ORGANIZATION_BLOCK "SYS_OBNL_FLT"	// OB 85
TITLE = "Organization Block (OB) Not Loaded Fault"
//COPYRIGHT:    (C) 2000 BY  BUHLER LTD.
//                           CH-9240 UZWIL  SWITZERLAND
//
//PRODUCT:      PROJECT    
//
//TITLE:        Priority Class Error Organization Block (OB85)
//             
//
//--------------------------------------------------------------------------------
//
//IDENT:        AUTOR:              DEPT:                            DATE:
//STD_OB85.2.1  A.Egli              CT3                              23-Nov-2004
//              Only no stop when I/O access error updating the process image
//STD_OB85.2.0  A.Egli              CT3                              12-Jul-2004
//              LOG Message
//STD_OB85.1.0  A.Egli              CT3                              05-Nov-2002
//              1st Release
//
//--------------------------------------------------------------------------------
//
//PURPOSE:      
//
//RESTRICTIONS:
//
//--------------------------------------------------------------------------------
//
AUTHOR : EA
FAMILY : ASW
NAME : OBNLFLT
VERSION : 2.1
VAR_TEMP
  OB85_EV_CLASS : BYTE ;	//16#35 Event class 3
  OB85_FLT_ID : BYTE ;	//16#XX, Fault identification code
  OB85_PRIORITY : BYTE ;	//26 (Priority of 1 is lowest)
  OB85_OB_NUMBR : BYTE ;	//85 (Organization block 85, OB85)
  OB85_RESERVED_1 : BYTE ;	//Reserved for system
  OB85_RESERVED_2 : BYTE ;	//Reserved for system
  OB85_RESERVED_3 : INT ;	//Reserved for system
  OB85_ERR_EV_NUM : BYTE ;	//Number of event causing error
  OB85_ERR_EV_CLASS : BYTE ;	//Class of event causing error
  OB85_OB_PRIOR : BYTE ;	//Priority of OB causing error
  OB85_OB_NUM : BYTE ;	//Number of OB causing error
  OB85_DATE_TIME : DATE_AND_TIME ;	//Date and time OB85 started
  tmpHeader : WORD ;
  tmpObjNo : WORD ;	//OB-Nummer [80..121]
  EVClass_FLTID : WORD ;	//EV_Class / FLT_ID
  tmpPara3 : WORD ;
  tmpPara4 : WORD ;
  tmpPara5 : WORD ;
  tmpPara6 : WORD ;	//---
  tmpPara7 : WORD ;	//---
  tmpPara8 : WORD ;	//---
  tmpDate : WORD ;
  tmpYearMonth : WORD ;
  tmpDayHour : WORD ;
  tmpMinSec : WORD ;
  tmp_Z23 : DWORD ;
  tmpNoStop : BOOL ;
END_VAR
BEGIN
NETWORK
TITLE =
NETWORK
TITLE = Log Message: Header
//Header
      A(;
      L     #OB85_EV_CLASS;
      L     B#16#34;	// going
      ==I;
      );
      JCN   komm;
      L     3;
      JU    tran;
komm: L     1;	// coming
tran: SLW   5;
      +     11;	// NEW MessageFormatNo
      T     #tmpHeader;
NETWORK
TITLE = Log Message: Para1 = Object Number
//--System Message---
      L     85;
      T     #tmpObjNo;
NETWORK
TITLE = Log Message: Para2 to 11
////
//Para2: EV_Class / FLT_ID
      L     #OB85_FLT_ID;
      L     W#16#FF;	// Only Low Byte
      AW;
      L     #OB85_EV_CLASS;
      SLD   8;
      OW;
      T     #EVClass_FLTID;
//Para3: Depending on fault identification code
      L     #OB85_OB_NUMBR;
      T     #tmpPara3;
//Para4: DKZ23
      L     #OB85_RESERVED_1;
      T     #tmpPara4;
//Para5: Z1
      L     #OB85_RESERVED_3;
      T     #tmpPara5;
//Para6: Z23 HW
      LAR1  P##OB85_ERR_EV_NUM;
      L     LW [AR1,P#0.0];
      T     #tmpPara6;
//Para7: Z23 LW
      L     LW [AR1,P#2.0];
      T     #tmpPara7;
//Para9 to 11: Date/Time
      LAR1  P##OB85_DATE_TIME;
      L     LB [AR1,P#0.0];
      BTI;
      SLD   8;
      L     LB [AR1,P#1.0];
      BTI;
      OW;
      T     #tmpYearMonth;
      L     LB [AR1,P#2.0];
      BTI;
      SLD   8;
      L     LB [AR1,P#3.0];
      BTI;
      OW;
      T     #tmpDayHour;
      L     LB [AR1,P#4.0];
      BTI;
      SLD   8;
      L     LB [AR1,P#5.0];
      BTI;
      OW;
      T     #tmpMinSec;
NETWORK
TITLE = Faults without STOP
// // alle auskommentierten Einträge führen in STOP
//
//B1,B2,B3,B4: I/O access error when updating the process image
      A(;
      L     B#16#F0;
      L     #OB85_FLT_ID;
      AW;
      L     B#16#B0;
      ==I;
      );
      =     #tmpNoStop;
NETWORK
TITLE = Log Message: Entry
//Entre Log Message
      AN    #tmpNoStop;
      S     "SYS_LOG_Queue".CmdAddFastMsg;
      CALL  "SYS_LOG_EntryQueue" (
           DBNumber                 := 5,
           Header                   := #tmpHeader,
           Para1                    := #tmpObjNo,
           Para2                    := #EVClass_FLTID,
           Para3                    := #tmpPara3,
           Para4                    := #tmpPara4,
           Para5                    := #tmpPara5,
           Para6                    := #tmpPara6,
           Para7                    := #tmpPara7,
           Para8                    := W#16#0,
           Para9                    := #tmpYearMonth,
           Para10                   := #tmpDayHour,
           Para11                   := #tmpMinSec);	//Header / Para1: ObjectNo / Para2: Class / FLTID / Para3: OB Number / Para4: DKZ23 / Para5: Z1 / Para6: Z23 HW / Para7: Z23 LW / Para8:  / Para9:  Year / Month / Para10: Day  / Hour / Para11: Min  / Sec 
NETWORK
TITLE = Stop PLC
      A     #tmpNoStop;
      BEC;
//**********************
// Bring CPU to Stop
      CALL  "SIEMENS_STP";
//**********************
NETWORK
TITLE = End of block
      BE;
END_ORGANIZATION_BLOCK

ORGANIZATION_BLOCK "SYS_RACK_FLT"	// OB 86
TITLE = "Loss Of Rack Fault"
//COPYRIGHT:    (C) 2000 BY  BUHLER AG
//                           CH-9240 UZWIL  SWITZERLAND
//
//PRODUCT:      PROJECT
//
//TITLE:        Loss of rack fault
//               Extended rack faults
//               DP-Master or slave faults
//              Erweiterungsgerätanschaltungsfehler
//               Erweiterungsgerätefehler
//               Profibus-DB Master- und Slavefehler
//
//--------------------------------------------------------------------------------
//IDENT:        AUTHOR:             DEPT:                             DATE:
//
//Pxx_OB086.2.0 A.Egli              CT3                               12-Jul-2004
//              Log message added
//Pxx_OB086.1.0 Ph. Engler          MU664                             16-Jan-2002
//              1st Release
//
//--------------------------------------------------------------------------------
//
//PURPOSE:      
//
//RESTRICTIONS: 
//
//--------------------------------------------------------------------------------
//
AUTHOR : EA
FAMILY : ASW
NAME : RACKFLT
VERSION : 2.0
VAR_TEMP
  OB86_EV_CLASS : BYTE ;	//16#38/39 Event class 3
  OB86_FLT_ID : BYTE ;	//16#C1/C4/C5, Fault identification code
  OB86_PRIORITY : BYTE ;	//26/28 (Priority of 1 is lowest)
  OB86_OB_NUMBR : BYTE ;	//86 (Organization block 86, OB86)
  OB86_RESERVED_1 : BYTE ;	//Reserved for system
  OB86_RESERVED_2 : BYTE ;	//Reserved for system
  OB86_MDL_ADDR : WORD ;	//Depending on fault identification code
  OB86_RACKS_FLTD : ARRAY  [0 .. 31 ] OF BOOL ;	//Racks in fault
  OB86_DATE_TIME : DATE_AND_TIME ;	//Date and time OB86 started
  tmpHeader : WORD ;
  tmpObjNo : WORD ;	//OB-Nummer [80..121]
  EVClass_FLTID : WORD ;	//EV_Class / FLT_ID
  tmpPara3 : WORD ;	//
  tmpPara4 : WORD ;	//
  tmpPara5 : WORD ;	//
  tmpPara6 : WORD ;	//
  tmpPara7 : WORD ;	//
  tmpDate : WORD ;
  tmpYearMonth : WORD ;
  tmpDayHour : WORD ;
  tmpMinSec : WORD ;
  tmp_Z23 : DWORD ;
  tmpSlave : INT ;
  tmpMaster : INT ;
  tmpNoStop : BOOL ;
END_VAR
BEGIN
NETWORK
TITLE = Detailed Diagnosis in OB86 (interrupt)
      CALL  "SYS_DPDiagMain";
NETWORK
TITLE = Log Message: Header
//Header
      A(;
      L     #OB86_EV_CLASS;
      L     B#16#38;	// going
      ==I;
      );
      JCN   komm;
      L     3;
      JU    tran;
komm: L     1;	// coming
tran: SLW   5;
      +     11;	// NEW MessageFormatNo
      T     #tmpHeader;
NETWORK
TITLE = Log Message: Para1 = Object Number
//Para1: Object Number
      LAR1  P##OB86_RACKS_FLTD;
      L     LD [AR1,P#0.0];
      T     #tmp_Z23;
      L     #tmp_Z23;
      SRD   8;
      L     DW#16#FF;
      AW;
      L     1000;
      *I;
      T     #tmpMaster;
      L     #tmp_Z23;
      L     DW#16#FF;
      AW;
      T     #tmpSlave;
//--DP Rack -----
      L     #OB86_FLT_ID;
      L     B#16#C1;
      ==I;
      JC    OJRA;
      L     #OB86_FLT_ID;
      L     B#16#C2;
      ==I;
      JC    OJRA;
      L     #OB86_FLT_ID;
      L     B#16#C6;
      ==I;
      JC    OJRA;
      JU    OJC3;
OJRA: LAR1  P##OB86_RACKS_FLTD;
//    Check Bit 1..21 of OB86_Racks_FLTD
      L     10001;
      T     #tmpObjNo;
OJR2: A     L [AR1,P#0.1];
      JC    OJJO;
      +AR1  P#0.1;
      L     121;
      L     #tmpObjNo;
      <=I;
      JC    OJR2;
      JU    OJSM;	//-->Illegal RackNr-->  Print as System message
//--DP Master -----
OJC3: L     #OB86_FLT_ID;
      L     B#16#C3;
      ==I;
      JC    OJMA;
      JU    OJC4;
OJMA: L     #tmpMaster;
      T     #tmpObjNo;
      JU    OJJO;
//---DP Station----
OJC4: L     #OB86_FLT_ID;
      L     B#16#C4;
      ==I;
      JC    OJSL;
      L     #OB86_FLT_ID;
      L     B#16#C5;
      ==I;
      JC    OJSL;
      L     #OB86_FLT_ID;
      L     B#16#C7;
      ==I;
      JC    OJSL;
      L     #OB86_FLT_ID;
      L     B#16#C8;
      ==I;
      JC    OJSL;
      JU    OJSM;
OJSL: L     #tmpMaster;
      L     #tmpSlave;
      +I;
      T     #tmpObjNo;
      JU    OJJO;
//--System Message---
OJSM: L     86;
      T     #tmpObjNo;
OJJO: NOP   0;
NETWORK
TITLE = Log Message: Para2 to 11
////
//Para2: EV_Class / FLT_ID
      L     #OB86_FLT_ID;
      L     W#16#FF;	// Only Low Byte
      AW;
      L     #OB86_EV_CLASS;
      SLD   8;
      OW;
      T     #EVClass_FLTID;
//Para3: Depending on fault identification code
      L     #OB86_OB_NUMBR;
      T     #tmpPara3;
//Para4:not used
      L     0;
      T     #tmpPara4;
//Para5: MDL_ADDR
      L     #OB86_MDL_ADDR;
      T     #tmpPara5;
//Para6: Z23 HW
      LAR1  P##OB86_RACKS_FLTD;
      L     LW [AR1,P#0.0];
      T     #tmpPara6;
//Para7: Z23 LW
      L     LW [AR1,P#2.0];
      T     #tmpPara7;
//Para9 to 11: Date/Time
      LAR1  P##OB86_DATE_TIME;
      L     LB [AR1,P#0.0];
      BTI;
      SLD   8;
      L     LB [AR1,P#1.0];
      BTI;
      OW;
      T     #tmpYearMonth;
      L     LB [AR1,P#2.0];
      BTI;
      SLD   8;
      L     LB [AR1,P#3.0];
      BTI;
      OW;
      T     #tmpDayHour;
      L     LB [AR1,P#4.0];
      BTI;
      SLD   8;
      L     LB [AR1,P#5.0];
      BTI;
      OW;
      T     #tmpMinSec;
NETWORK
TITLE = Faults without STOP
// // alle auskommentierten Einträge führen in STOP
//
// C1 Expansion rack failure
      O(;
      L     #OB86_FLT_ID;
      L     B#16#C1;	// 
      ==I;
      );
// C2 Expansion rack operational again
      O(;
      L     #OB86_FLT_ID;
      L     B#16#C2;	// 
      ==I;
      );
// C3 Failure of  DP master
      O(;
      L     #OB86_FLT_ID;
      L     B#16#C3;	// 
      ==I;
      );
// C4 Failure of DP Slave
      O(;
      L     #OB86_FLT_ID;
      L     B#16#C4;	// 
      ==I;
      );
// C5 Fault in a DP Slave
      O(;
      L     #OB86_FLT_ID;
      L     B#16#C5;	// 
      ==I;
      );
// C6 Expansion rack with error in module parameter
      O(;
      L     #OB86_FLT_ID;
      L     B#16#C6;	// 
      ==I;
      );
// C7 Return DP Slave with error in modul parameter
      O(;
      L     #OB86_FLT_ID;
      L     B#16#C7;	// 
      ==I;
      );
// C8 DP Slave configuartion <> actual configuration
      O(;
      L     #OB86_FLT_ID;
      L     B#16#C8;	// 
      ==I;
      );
      =     #tmpNoStop;
NETWORK
TITLE = Log Message: Entry
//Entre Log Message
      AN    #tmpNoStop;
      S     "SYS_LOG_Queue".CmdAddFastMsg;
      CALL  "SYS_LOG_EntryQueue" (
           DBNumber                 := 5,
           Header                   := #tmpHeader,
           Para1                    := #tmpObjNo,
           Para2                    := #EVClass_FLTID,
           Para3                    := #tmpPara3,
           Para4                    := W#16#0,
           Para5                    := #tmpPara5,
           Para6                    := #tmpPara6,
           Para7                    := #tmpPara7,
           Para8                    := W#16#0,
           Para9                    := #tmpYearMonth,
           Para10                   := #tmpDayHour,
           Para11                   := #tmpMinSec);	//Header / Para1: ObjectNo / Para2: Class / FLTID / Para3: OB Number / Para4: / Para5: MDL_ADDR / Para6: Z23 HW / Para7: Z23 HW / Para8:  / Para9:  Year / Month / Para10: Day  / Hour / Para11: Min  / Sec 
NETWORK
TITLE = Stop PLC
      A     #tmpNoStop;
      BEC;
//**********************
// Bring CPU to Stop
      CALL  "SIEMENS_STP";
//**********************
NETWORK
TITLE = End of block
      BE;
END_ORGANIZATION_BLOCK

ORGANIZATION_BLOCK "PLC_StUpNewstart"	// OB 100
TITLE = Startup program on newstart
//COPYRIGHT:    (C) 2000 BY  BUHLER AG
//                           CH-9240 UZWIL  SWITZERLAND
//
//PRODUCT:      PROJECT
//
//TITLE:        Startup program on newstart
//              
//              Anlaufprogramm bei Neustart
//
//
//--------------------------------------------------------------------------------
//
//IDENT:        AUTHOR:             DEPT:                             DATE:
//
//Pxx_OB102.2.0 A.Egli              CT3                               15-Jul-2004
//              Log Message
//Pxx_OB100.1.0 Ph. Engler          MU664                             05-Jan-2000
//              1st Release
//
//--------------------------------------------------------------------------------
//
//PURPOSE:      
//
//RESTRICTIONS: 
//
//--------------------------------------------------------------------------------
//
AUTHOR : PE
FAMILY : ASW
NAME : StUpNew
VERSION : 2.0
VAR_TEMP
  OB100_EV_CLASS : BYTE ;	//16#13, Event class 1, Entering event state, Event logged in diagnostic buffer
  OB100_STRTUP : BYTE ;	//16#81/82/83/84 Method of startup
  OB100_PRIORITY : BYTE ;	//27 (Priority of 1 is lowest)
  OB100_OB_NUMBR : BYTE ;	//100 (Organization block 100, OB100)
  OB100_RESERVED_1 : BYTE ;	//Reserved for system
  OB100_RESERVED_2 : BYTE ;	//Reserved for system
  OB100_STOP : WORD ;	//Event that caused CPU to stop (16#4xxx)
  OB100_STRT_INFO : DWORD ;	//Information on how system started
  OB100_DATE_TIME : DATE_AND_TIME ;	//Date and time OB100 started
  tmpHeader : WORD ;
  tmpObjNo : WORD ;	//OB-Nummer [80..121]
  EVClass_FLTID : WORD ;	//EV_Class / FLT_ID
  tmpPara3 : WORD ;	//
  tmpDate : WORD ;
  tmpYearMonth : WORD ;
  tmpDayHour : WORD ;
  tmpMinSec : WORD ;
END_VAR
BEGIN
NETWORK
TITLE = Create startup signals
      L     #OB100_STRTUP;
      L     B#16#81;
      ==I;
      S     "PLC_SystemDB".Startup.CmdNewstartMan;
      L     #OB100_STRTUP;
      L     B#16#82;
      ==I;
      S     "PLC_SystemDB".Startup.CmdNewstartAuto;
NETWORK
TITLE = Startup counters
      AN    "PLC_SystemDB".Startup.CmdNewstartMan;
      JC    n2n1;
      L     "PLC_SystemDB".StartupCounter.NewstartMan;
      +     1;
      T     "PLC_SystemDB".StartupCounter.NewstartMan;
      JU    n2e;
n2n1: AN    "PLC_SystemDB".Startup.CmdNewstartAuto;
      JC    n2e;
      L     "PLC_SystemDB".StartupCounter.NewstartAuto;
      +     1;
      T     "PLC_SystemDB".StartupCounter.NewstartAuto;
n2e:  NOP   0;
NETWORK
TITLE = General plc startup functions
      CALL  "SYS_GeneralPLCStartup";
NETWORK
TITLE = Special plant startup functions
NETWORK
TITLE = Reset startup flags
      SET;
      R     "PLC_SystemDB".Startup.CmdNewstartMan;
      R     "PLC_SystemDB".Startup.CmdNewstartAuto;
NETWORK
TITLE = Log Message: Header
//Header
      L     3;	// Operator
      SLW   5;
      +     11;	// NEW MessageFormatNo
      T     #tmpHeader;
NETWORK
TITLE = Log Message: Para1 = Object Number
//Para1: Object Number
//--System Message---
      L     #OB100_OB_NUMBR;
      T     #tmpObjNo;
NETWORK
TITLE = Log Message: Para2 to 11
////
//Para2: EV_Class / FLT_ID
      L     #OB100_STRTUP;
      L     W#16#FF;	// Only Low Byte
      AW;
      L     #OB100_EV_CLASS;
      SLD   8;
      OW;
      T     #EVClass_FLTID;
//Para3: Depending on fault identification code
      L     #OB100_OB_NUMBR;
      T     #tmpPara3;
//Para9 to 11: Date/Time
      LAR1  P##OB100_DATE_TIME;
      L     LB [AR1,P#0.0];
      BTI;
      SLD   8;
      L     LB [AR1,P#1.0];
      BTI;
      OW;
      T     #tmpYearMonth;
      L     LB [AR1,P#2.0];
      BTI;
      SLD   8;
      L     LB [AR1,P#3.0];
      BTI;
      OW;
      T     #tmpDayHour;
      L     LB [AR1,P#4.0];
      BTI;
      SLD   8;
      L     LB [AR1,P#5.0];
      BTI;
      OW;
      T     #tmpMinSec;
NETWORK
TITLE = Log Message: Entry
//Entre Log Message
      CALL  "SYS_LOG_EntryQueue" (
           DBNumber                 := 5,
           Header                   := #tmpHeader,
           Para1                    := #tmpObjNo,
           Para2                    := #EVClass_FLTID,
           Para3                    := #tmpPara3,
           Para4                    := W#16#0,
           Para5                    := W#16#0,
           Para6                    := W#16#0,
           Para7                    := W#16#0,
           Para8                    := W#16#0,
           Para9                    := #tmpYearMonth,
           Para10                   := #tmpDayHour,
           Para11                   := #tmpMinSec);	//Header / Para1: ObjectNo / Para2: Class / STRTUP / Para3: OB Number / Para4: / Para5:  / Para6:  / Para7: / Para8:  / Para9:  Year / Month / Para10: Day  / Hour / Para11: Min  / Sec 
NETWORK
TITLE = End of block
      BE;
END_ORGANIZATION_BLOCK

ORGANIZATION_BLOCK "PLC_StUpRestart"	// OB 101
TITLE = Startup program on restart
//COPYRIGHT:    (C) 2000 BY  BUHLER AG
//                           CH-9240 UZWIL  SWITZERLAND
//
//PRODUCT:      PROJECT
//
//TITLE:        Startup program on restart
//                 After voltage returned
//              Anlaufprogramm  bei Wiederanlauf
//                 Nach Spannungswiederkehr
//
//--------------------------------------------------------------------------------
//
//IDENT:        AUTHOR:             DEPT:                             DATE:
//
//Pxx_OB101.3.0 A.Egli              CT3                               15-Jul-2004
//              The following lines are moved to OB1
//                R     "PLC_SystemDB".Startup.CmdRestartMan
//                R     "PLC_SystemDB".Startup.CmdRestartAuto
//Pxx_OB101.2.0 A.Egli              CT3                               15-Jul-2004
//              Log Message
//Pxx_OB101.1.0 Ph. Engler          MU664                             05-Jan-2000
//              1st Release
//
//--------------------------------------------------------------------------------
//
//PURPOSE:      
//
//RESTRICTIONS: 
//
//--------------------------------------------------------------------------------
//
AUTHOR : PE
FAMILY : ASW
NAME : StUpRest
VERSION : 3.0
VAR_TEMP
  OB101_EV_CLASS : BYTE ;	//16#13, Event class 1, Entering event state, Event logged in diagnostic buffer
  OB101_STRTUP : BYTE ;	//16#81/82/83/84 Method of startup
  OB101_PRIORITY : BYTE ;	//27 (Priority of 1 is lowest)
  OB101_OB_NUMBR : BYTE ;	//101 (Organization block 101, OB101)
  OB101_RESERVED_1 : BYTE ;	//Reserved for system
  OB101_RESERVED_2 : BYTE ;	//Reserved for system
  OB101_STOP : WORD ;	//Event that caused CPU to stop (16#4xxx)
  OB101_STRT_INFO : DWORD ;	//Information on how system started
  OB101_DATE_TIME : DATE_AND_TIME ;	//Date and time OB101 started
  tmpHeader : WORD ;
  tmpObjNo : WORD ;	//OB-Nummer [80..121]
  EVClass_FLTID : WORD ;	//EV_Class / FLT_ID
  tmpPara3 : WORD ;	//
  tmpDate : WORD ;
  tmpYearMonth : WORD ;
  tmpDayHour : WORD ;
  tmpMinSec : WORD ;
END_VAR
BEGIN
NETWORK
TITLE = Create startup flags
      L     #OB101_STRTUP;
      L     B#16#83;
      ==I;
      S     "PLC_SystemDB".Startup.CmdRestartMan;
      L     #OB101_STRTUP;
      L     B#16#84;
      ==I;
      S     "PLC_SystemDB".Startup.CmdRestartAuto;
NETWORK
TITLE = Startup counters
      AN    "PLC_SystemDB".Startup.CmdRestartMan;
      JC    n2n1;
      L     "PLC_SystemDB".StartupCounter.RestartMan;
      +     1;
      T     "PLC_SystemDB".StartupCounter.RestartMan;
      JU    n2e;
n2n1: AN    "PLC_SystemDB".Startup.CmdRestartAuto;
      JC    n2e;
      L     "PLC_SystemDB".StartupCounter.RestartAuto;
      +     1;
      T     "PLC_SystemDB".StartupCounter.RestartAuto;
n2e:  NOP   0;
NETWORK
TITLE = General plc startup functions
      CALL  "SYS_GeneralPLCStartup";
NETWORK
TITLE = Special plant startup functions
NETWORK
TITLE = Reset startup flags
//[3.0]      SET   
//[3.0]      R     "PLC_SystemDB".Startup.CmdRestartMan
//[3.0]      R     "PLC_SystemDB".Startup.CmdRestartAuto
NETWORK
TITLE = Log Message: Header
//Header
      L     3;	// Operator
      SLW   5;
      +     11;	// NEW MessageFormatNo
      T     #tmpHeader;
NETWORK
TITLE = Log Message: Para1 = Object Number
//Para1: Object Number
//--System Message---
      L     #OB101_OB_NUMBR;
      T     #tmpObjNo;
NETWORK
TITLE = Log Message: Para2 to 11
////
//Para2: EV_Class / FLT_ID
      L     #OB101_STRTUP;
      L     W#16#FF;	// Only Low Byte
      AW;
      L     #OB101_EV_CLASS;
      SLD   8;
      OW;
      T     #EVClass_FLTID;
//Para3: Depending on fault identification code
      L     #OB101_OB_NUMBR;
      T     #tmpPara3;
//Para9 to 11: Date/Time
      LAR1  P##OB101_DATE_TIME;
      L     LB [AR1,P#0.0];
      BTI;
      SLD   8;
      L     LB [AR1,P#1.0];
      BTI;
      OW;
      T     #tmpYearMonth;
      L     LB [AR1,P#2.0];
      BTI;
      SLD   8;
      L     LB [AR1,P#3.0];
      BTI;
      OW;
      T     #tmpDayHour;
      L     LB [AR1,P#4.0];
      BTI;
      SLD   8;
      L     LB [AR1,P#5.0];
      BTI;
      OW;
      T     #tmpMinSec;
NETWORK
TITLE = Log Message: Entry
//Entre Log Message
      CALL  "SYS_LOG_EntryQueue" (
           DBNumber                 := 5,
           Header                   := #tmpHeader,
           Para1                    := #tmpObjNo,
           Para2                    := #EVClass_FLTID,
           Para3                    := #tmpPara3,
           Para4                    := W#16#0,
           Para5                    := W#16#0,
           Para6                    := W#16#0,
           Para7                    := W#16#0,
           Para8                    := W#16#0,
           Para9                    := #tmpYearMonth,
           Para10                   := #tmpDayHour,
           Para11                   := #tmpMinSec);	//Header / Para1: ObjectNo / Para2: Class / STRTUP / Para3: OB Number / Para4: / Para5:  / Para6:  / Para7: / Para8:  / Para9:  Year / Month / Para10: Day  / Hour / Para11: Min  / Sec 
NETWORK
TITLE = End of block
      BE;
END_ORGANIZATION_BLOCK

ORGANIZATION_BLOCK "PLC_StUpColdstart"	// OB 102
TITLE = Startup program on coldstart
//COPYRIGHT:    (C) 2000 BY  BUHLER AG
//                           CH-9240 UZWIL  SWITZERLAND
//
//PRODUCT:      PROJECT
//
//TITLE:        Startup program on coldstart
//              
//              Anlaufprogramm bei Kaltstart
//
//
//--------------------------------------------------------------------------------
//
//IDENT:        AUTHOR:             DEPT:                             DATE:
//
//Pxx_OB102.2.0 A.Egli              CT3                               15-Jul-2004
//              Log Message
//Pxx_OB102.1.0 Ph. Engler          MU664                             17-Dez-2000
//              1st Release
//
//--------------------------------------------------------------------------------
//
//PURPOSE:      
//
//RESTRICTIONS: 
//
//--------------------------------------------------------------------------------
//
AUTHOR : PE
FAMILY : ASW
NAME : StUpCold
VERSION : 2.0
VAR_TEMP
  OB102_EV_CLASS : BYTE ;	//16#13, Event class 1, Entering event state, Event logged in diagnostic buffer
  OB102_STRTUP : BYTE ;	//16#85...8B Method of startup
  OB102_PRIORITY : BYTE ;	//27 (Priority of 1 is lowest)
  OB102_OB_NUMBR : BYTE ;	//102 (Organization block 102, OB102)
  OB102_RESERVED_1 : BYTE ;	//Reserved for system
  OB102_RESERVED_2 : BYTE ;	//Reserved for system
  OB102_STOP : WORD ;	//Event that caused CPU to stop (16#4xxx)
  OB102_STRT_INFO : DWORD ;	//Information on how system started
  OB102_DATE_TIME : DATE_AND_TIME ;	//Date and time OB102 started
  tmpHeader : WORD ;
  tmpObjNo : WORD ;	//OB-Nummer [80..121]
  EVClass_FLTID : WORD ;	//EV_Class / FLT_ID
  tmpPara3 : WORD ;	//
  tmpDate : WORD ;
  tmpYearMonth : WORD ;
  tmpDayHour : WORD ;
  tmpMinSec : WORD ;
END_VAR
BEGIN
NETWORK
TITLE = Create startup signals
      L     #OB102_STRTUP;
      L     B#16#85;
      ==I;
      S     "PLC_SystemDB".Startup.CmdColdstartMan;
// 
      L     #OB102_STRTUP;
      L     B#16#86;
      ==I;
      S     "PLC_SystemDB".Startup.CmdColdstartAuto;
NETWORK
TITLE = Startup counters
      AN    "PLC_SystemDB".Startup.CmdColdstartMan;
      JC    n2n1;
      L     "PLC_SystemDB".StartupCounter.ColdstartMan;
      +     1;
      T     "PLC_SystemDB".StartupCounter.ColdstartMan;
      JU    n2e;
n2n1: AN    "PLC_SystemDB".Startup.CmdColdstartAuto;
      JC    n2e;
      L     "PLC_SystemDB".StartupCounter.ColdstartAuto;
      +     1;
      T     "PLC_SystemDB".StartupCounter.ColdstartAuto;
n2e:  NOP   0;
NETWORK
TITLE = General plc startup functions
      CALL  "SYS_GeneralPLCStartup";
NETWORK
TITLE = Special plant startup functions
NETWORK
TITLE = Reset startup flags
      SET;
      R     "PLC_SystemDB".Startup.CmdColdstartMan;
      R     "PLC_SystemDB".Startup.CmdColdstartAuto;
NETWORK
TITLE = Log Message: Header
//Header
      L     3;	// Operator
      SLW   5;
      +     11;	// NEW MessageFormatNo
      T     #tmpHeader;
NETWORK
TITLE = Log Message: Para1 = Object Number
//Para1: Object Number
//--System Message---
      L     #OB102_OB_NUMBR;
      T     #tmpObjNo;
NETWORK
TITLE = Log Message: Para2 to 11
////
//Para2: EV_Class / FLT_ID
      L     #OB102_STRTUP;
      L     W#16#FF;	// Only Low Byte
      AW;
      L     #OB102_EV_CLASS;
      SLD   8;
      OW;
      T     #EVClass_FLTID;
//Para3: Depending on fault identification code
      L     #OB102_OB_NUMBR;
      T     #tmpPara3;
//Para9 to 11: Date/Time
      LAR1  P##OB102_DATE_TIME;
      L     LB [AR1,P#0.0];
      BTI;
      SLD   8;
      L     LB [AR1,P#1.0];
      BTI;
      OW;
      T     #tmpYearMonth;
      L     LB [AR1,P#2.0];
      BTI;
      SLD   8;
      L     LB [AR1,P#3.0];
      BTI;
      OW;
      T     #tmpDayHour;
      L     LB [AR1,P#4.0];
      BTI;
      SLD   8;
      L     LB [AR1,P#5.0];
      BTI;
      OW;
      T     #tmpMinSec;
NETWORK
TITLE = Log Message: Entry
//Entre Log Message
      CALL  "SYS_LOG_EntryQueue" (
           DBNumber                 := 5,
           Header                   := #tmpHeader,
           Para1                    := #tmpObjNo,
           Para2                    := #EVClass_FLTID,
           Para3                    := #tmpPara3,
           Para4                    := W#16#0,
           Para5                    := W#16#0,
           Para6                    := W#16#0,
           Para7                    := W#16#0,
           Para8                    := W#16#0,
           Para9                    := #tmpYearMonth,
           Para10                   := #tmpDayHour,
           Para11                   := #tmpMinSec);	//Header / Para1: ObjectNo / Para2: Class / STRTUP / Para3: OB Number / Para4: / Para5:  / Para6:  / Para7: / Para8:  / Para9:  Year / Month / Para10: Day  / Hour / Para11: Min  / Sec 
NETWORK
TITLE = End of block
      BE;
END_ORGANIZATION_BLOCK

ORGANIZATION_BLOCK "SYS_PROG_ERR"	// OB 121
//COPYRIGHT:    (C) 2000 BY  BUHLER AG
//                           CH-9240 UZWIL  SWITZERLAND
//
//PRODUCT:      PROJECT
//
//TITLE:        OB121 
//              
//
//--------------------------------------------------------------------------------
//IDENT:        AUTHOR:             DEPT:                             DATE:
//
//OB121.2.0     A.Egli              CT3                               13-Jul-2004
//              1st Release
//OB121.1A      TIK                 MU664                             13-Apr-99
//              1st Release
//OB121.1B      Tho                 FU53                              16-Dez-99
//              FU-Version erstellt 
//
//--------------------------------------------------------------------------------
//
//PURPOSE:      
//
//RESTRICTIONS: 
//
//--------------------------------------------------------------------------------
//
AUTHOR : EA
FAMILY : ASW
NAME : PROG_ERR
VERSION : 2.0
VAR_TEMP
  OB121_EV_CLASS : BYTE ;	//16#25, Event class 2, Entering event state, Internal fault event
  OB121_SW_FLT : BYTE ;	//16#XX Software programming fault
  OB121_PRIORITY : BYTE ;	//X = Priority of OB where fault occured (Priority of 1 is lowest)
  OB121_OB_NUMBR : BYTE ;	//121 (Organization block 121, OB121)
  OB121_BLK_TYPE : BYTE ;	//16#88/8A/8B/8C/8E Type of block fault occured in
  OB121_RESERVED_1 : BYTE ;	//Reserved for system
  OB121_FLT_REG : WORD ;	//16#XX Specific register that caused fault
  OB121_BLK_NUM : WORD ;	//Number of block that programming fault occured in
  OB121_PRG_ADDR : WORD ;	//Address in block where programming fault occured
  OB121_DATE_TIME : DATE_AND_TIME ;	//Date and time OB121 started
  tmpHeader : WORD ;
  tmpObjNo : WORD ;	//OB-Nummer [80..121]
  EVClass_FLTID : WORD ;	//EV_Class / FLT_ID
  tmpPara3 : WORD ;	//Reserved 1 for system
  tmpPara4 : WORD ;	//Input module (01010100), Output module (01010101)
  tmpPara5 : WORD ;	//Base address of module with point fault
  tmpPara6 : WORD ;	//Module type with point fault
  tmpPara7 : WORD ;	//Module type with point fault
  tmpYearMonth : WORD ;
  tmpDayHour : WORD ;
  tmpMinSec : WORD ;
  tmpNoStop : BOOL ;
END_VAR
BEGIN
NETWORK
TITLE =
NETWORK
TITLE = Log Message: Header
      A(;
      L     #OB121_EV_CLASS;
      L     B#16#38;	// going
      ==I;
      );
      JCN   komm;
      L     3;
      JU    tran;
komm: L     1;	// coming
tran: SLW   5;
      +     11;	// NEW MessageFormatNo
      T     #tmpHeader;
NETWORK
TITLE = Log Message: Para1 = Object Number
//--System Message---
      L     121;
      T     #tmpObjNo;
NETWORK
TITLE = Log Message: Para2 to 11
////
//Para2: EV_Class / FLT_ID
      L     #OB121_SW_FLT;
      L     W#16#FF;	// Only Low Byte
      AW;
      L     #OB121_EV_CLASS;
      SLD   8;
      OW;
      T     #EVClass_FLTID;
//Para3: OB_NUMBR
      L     #OB121_OB_NUMBR;
      T     #tmpPara3;
//Para4: OB121_FLT_REG
      L     #OB121_FLT_REG;
      T     #tmpPara4;
//Para5: OB121_BLK_TYPE
      L     #OB121_BLK_TYPE;
      T     #tmpPara5;
//Para6: Number of block that programming fault occured in
      L     #OB121_BLK_NUM;
      T     #tmpPara6;
//Para7: Address in block where programming fault occured
      L     #OB121_PRG_ADDR;
      T     #tmpPara7;
//Para9 to 11: Date/Time
      LAR1  P##OB121_DATE_TIME;
      L     LB [AR1,P#0.0];
      BTI;
      SLD   8;
      L     LB [AR1,P#1.0];
      BTI;
      OW;
      T     #tmpYearMonth;
      L     LB [AR1,P#2.0];
      BTI;
      SLD   8;
      L     LB [AR1,P#3.0];
      BTI;
      OW;
      T     #tmpDayHour;
      L     LB [AR1,P#4.0];
      BTI;
      SLD   8;
      L     LB [AR1,P#5.0];
      BTI;
      OW;
      T     #tmpMinSec;
NETWORK
TITLE = Faults without STOP
//// alle auskommentierten Einträge führen in STOP 
//
      CLR;	//init.VKE  
// 21 BCD conversion error
      O(;
      L     #OB121_SW_FLT;
      L     B#16#21;	// 
      ==I;
      );
// 22 Area length error when reading
//      O(    
//      L     #OB121_SW_FLT
//      L     B#16#22                     // 
//      ==I   
//      )     
// 23 Range error when writing
//      O(    
//      L     #OB121_SW_FLT
//      L     B#16#23                     // 
//      ==I   
//      )     
// 24 Range access with pointer
//      O(    
//      L     #OB121_SW_FLT
//      L     B#16#24                     // 
//      ==I   
//      )     
// 25 Writing access with pointer
//      O(    
//      L     #OB121_SW_FLT
//      L     B#16#25                     // 
//      ==I   
//      )     
// 26 Error for timer number
//     O(    
//      L     #OB121_SW_FLT
//      L     B#16#26                     // 
//      ==I   
//      )     
// 27 Error for Counter
//      O(           
//      L     #OB121_SW_FLT
//      L     B#16#27                     // 
//      ==I   
//      )     
// 28  Reading access with pointer Bit<>0
//      O(    
//      L     #OB121_SW_FLT
//      L     B#16#28                     // 
//      ==I   
//      )     
// 29  Reading access with pointer Bit<>0
//      O(    
//      L     #OB121_SW_FLT
//      L     B#16#29                     // 
//      ==I   
//      )     
// 30 Write access GlobalDB
//      O(    
//      L     #OB121_SW_FLT
//      L     B#16#30                     // 
//      ==I   
//      )     
// 31 Write access InstanzDB
//      O(    
//      L     #OB121_SW_FLT
//      L     B#16#31                     // 
//     ==I   
//     )     
// 32 DB number GlobalDB
//      O(    
//      L     #OB121_SW_FLT
//      L     B#16#32                     // 
//      ==I   
//      )     
// 33 DB number InstanzDB
//      O(    
//      L     #OB121_SW_FLT
//      L     B#16#33                     // 
//      ==I   
//      )     
// 34 FC Number
//      O(    
//      L     #OB121_SW_FLT
//      L     B#16#34                     // 
//      ==I   
//      )     
// 35 FB Number
//      O(    
//      L     #OB121_SW_FLT
//      L     B#16#35                     // 
//      ==I   
//      )     
// 3A DB not loaded
//      O(    
//      L     #OB121_SW_FLT
//      L     B#16#3A                     // 
//      ==I   
//      )     
// 3C FC not loaded
//      O(    
//      L     #OB121_SW_FLT
//      L     B#16#3C                     // 
//      ==I   
//      )     
// 3D SFC not loaded
//      O(    
//      L     #OB121_SW_FLT
//      L     B#16#3D                     // 
//      ==I   
//      )     
// 3E FB not loaded
//      O(    
//      L     #OB121_SW_FLT
//      L     B#16#3E                     // 
//      ==I   
//      )     
// 3F SFB not loaded
//      O(    
//      L     #OB121_SW_FLT
//      L     B#16#3F                     // 
//      ==I   
//      )     
      =     #tmpNoStop;
NETWORK
TITLE = Log Message: Entry
//Log Meldung eintragen
      L     "SYS_LOG_Queue".VarNrOfMsgInQueue;
      L     0;
      <>I;
      A     #tmpNoStop;
      JC    LOJ0;
      AN    #tmpNoStop;
      S     "SYS_LOG_Queue".CmdAddFastMsg;
      CALL  "SYS_LOG_EntryQueue" (
           DBNumber                 := 5,
           Header                   := #tmpHeader,
           Para1                    := #tmpObjNo,
           Para2                    := #EVClass_FLTID,
           Para3                    := #tmpPara3,
           Para4                    := #tmpPara4,
           Para5                    := #tmpPara5,
           Para6                    := #tmpPara6,
           Para7                    := #tmpPara7,
           Para8                    := W#16#0,
           Para9                    := #tmpYearMonth,
           Para10                   := #tmpDayHour,
           Para11                   := #tmpMinSec);	//Header / Para1: ObjectNo / Para2: Class / FLTID / Para3: OB Number / Para4: FLT_REG / Para5: BLK_TYPE / Para6: BLK_NUM / Para7: PGR_ADDR / Para8:  / Para9:  Year / Month / Para10: Day  / Hour / Para11: Min  / Sec 
LOJ0: NOP   0;
NETWORK
TITLE = Stop PLC
      A     #tmpNoStop;
      BEC;
//**********************
// Bring CPU to Stop
      CALL  "SIEMENS_STP";
//**********************
NETWORK
TITLE = End of block
      BE;
END_ORGANIZATION_BLOCK

ORGANIZATION_BLOCK "SYS_MOD_ERR"	// OB 122
TITLE = "Module Access Error"
//COPYRIGHT:    (C) 2000 BY  BUHLER AG
//                           CH-9240 UZWIL  SWITZERLAND
//
//PRODUCT:      GEN_MU664
//
//TITLE:        Failure reading/wrinting to/from the peripherie
//
//              Peripheriezugriffsfehler
//              
//
//--------------------------------------------------------------------------------
//IDENT:        AUTHOR:             DEPT:                              DATE:
//
//GEN_OB122.2.0 Ph. Engler          MU664                              11-Feb-2003
//              Redesign GCS7 Release 2
//GEN_OB122.1.1 Ph. Engler          MU664                              22-Oct-2002
//              - MU test flag integrated
//GEN_OB122.1.0 A. Egli             CT3                                19-Oct-2002
//              1st Release
//
//--------------------------------------------------------------------------------
//
//PURPOSE:      
//
//RESTRICTIONS: 
//
//--------------------------------------------------------------------------------
//
AUTHOR : EA
FAMILY : SYS
NAME : SYS_ER
VERSION : 0.1
VAR_TEMP
  OB122_EV_CLASS : BYTE ;	//16#29, Event class 2, Entering event state, Internal fault event
  OB122_SW_FLT : BYTE ;	//16#XX Software error code
  OB122_PRIORITY : BYTE ;	//X = Priority of OB where fault occured (Priority of 1 is lowest)
  OB122_OB_NUMBR : BYTE ;	//122 (Organization block 122, OB122)
  OB122_BLK_TYPE : BYTE ;	//16#88/8A/8C/8E Type of block fault occured in
  OB122_MEM_AREA : BYTE ;	//Memory area where access error occured
  OB122_MEM_ADDR : WORD ;	//Memory address where access error occured
  OB122_BLK_NUM : WORD ;	//Block number in which error occured
  OB122_PRG_ADDR : WORD ;	//Program address where error occured
  OB122_DATE_TIME : DATE_AND_TIME ;	//Date and time OB1 started
  tmpAddr : DWORD ;
  tmpValue : DWORD ;
  tmpError : INT ;
END_VAR
BEGIN
NETWORK
TITLE = TM AS-Stop if no test mode
      AN    "PLC_SystemDB".TestFunctions.StaIOSimuli;
      ON    "PLC_SystemDB".GlobalFlags.StaTest;
      BEC;
NETWORK
TITLE = SI Simulation with DB16/DB17 or PA
      T     #tmpValue;
      AN    "GCS7_Gr_SimDPtoImage";
      JC    DBIO;
NETWORK
TITLE = PA Simulation with PA
      L     #OB122_MEM_AREA;
      L     2#111;
      AW;
      L     0;
      <>I;
      BEC;
      L     #OB122_MEM_ADDR;
      SLD   3;
      T     #tmpAddr;
      L     W#16#42;
      L     #OB122_SW_FLT;
      ==I;
      JC    Inp;
      L     W#16#44;
      L     #OB122_SW_FLT;
      ==I;
      JC    Inp;
      L     W#16#43;
      L     #OB122_SW_FLT;
      ==I;
      JC    Out1;
      L     W#16#45;
      L     #OB122_SW_FLT;
      ==I;
      JC    Out1;
      BEU;
Inp:  L     #OB122_MEM_AREA;
      SRW   4;
      L     1;
      <>I;
      JC    Inp2;
      L     IB [#tmpAddr];
      T     #tmpValue;
      CALL  "SIEMENS_REPL_VAL" (
           VAL                      := #tmpValue,
           RET_VAL                  := #tmpError);
      BEU;
Inp2: TAK;
      L     2;
      <>I;
      JC    Inp3;
      L     IW [#tmpAddr];
      T     #tmpValue;
      CALL  "SIEMENS_REPL_VAL" (
           VAL                      := #tmpValue,
           RET_VAL                  := #tmpError);
      BEU;
Inp3: TAK;
      L     3;
      <>I;
      BEC;
      L     ID [#tmpAddr];
      T     #tmpValue;
      CALL  "SIEMENS_REPL_VAL" (
           VAL                      := #tmpValue,
           RET_VAL                  := #tmpError);
      BEU;
Out1: L     #OB122_MEM_AREA;
      SRW   4;
      L     1;
      <>I;
      JC    Out2;
      L     #tmpValue;
      T     QB [#tmpAddr];
      BEU;
Out2: TAK;
      L     2;
      <>I;
      JC    Out3;
      L     #tmpValue;
      T     QW [#tmpAddr];
      BEU;
Out3: TAK;
      L     3;
      <>I;
      BEC;
      L     #tmpValue;
      T     QD [#tmpAddr];
      BEU;
NETWORK
TITLE =
DBIO: L     #OB122_MEM_AREA;
      L     2#111;
      AW;
      L     0;
      <>I;
      BEC;
      L     #OB122_MEM_ADDR;
      SLD   3;
      T     #tmpAddr;
      L     W#16#42;
      L     #OB122_SW_FLT;
      ==I;
      JC    IDB;
      L     W#16#44;
      L     #OB122_SW_FLT;
      ==I;
      JC    IDB;
      L     W#16#43;
      L     #OB122_SW_FLT;
      ==I;
      JC    ODB1;
      L     W#16#45;
      L     #OB122_SW_FLT;
      ==I;
      JC    ODB1;
      BEU;
IDB:  L     #OB122_MEM_AREA;
      SRW   4;
      L     1;
      <>I;
      JC    IDB2;
      OPN   "TEST_IOSimuliInput";
      L     DBB [#tmpAddr];
      T     #tmpValue;
      CALL  "SIEMENS_REPL_VAL" (
           VAL                      := #tmpValue,
           RET_VAL                  := #tmpError);
      BEU;
IDB2: TAK;
      L     2;
      <>I;
      JC    IDB3;
      OPN   "TEST_IOSimuliInput";
      L     DBW [#tmpAddr];
      T     #tmpValue;
      CALL  "SIEMENS_REPL_VAL" (
           VAL                      := #tmpValue,
           RET_VAL                  := #tmpError);
      BEU;
IDB3: TAK;
      L     3;
      <>I;
      BEC;
      OPN   "TEST_IOSimuliInput";
      L     DBD [#tmpAddr];
      T     #tmpValue;
      CALL  "SIEMENS_REPL_VAL" (
           VAL                      := #tmpValue,
           RET_VAL                  := #tmpError);
      BEU;
ODB1: L     #OB122_MEM_AREA;
      SRW   4;
      L     1;
      <>I;
      JC    ODB2;
      L     #tmpValue;
      OPN   "TEST_IOSimuliOutput";
      T     DBB [#tmpAddr];
      BEU;
ODB2: TAK;
      L     2;
      <>I;
      JC    ODB3;
      L     #tmpValue;
      OPN   "TEST_IOSimuliOutput";
      T     DBW [#tmpAddr];
      BEU;
ODB3: TAK;
      L     3;
      <>I;
      BEC;
      L     #tmpValue;
      OPN   "TEST_IOSimuliOutput";
      T     DBD [#tmpAddr];
      BEU;
NETWORK
TITLE = End of block
      BE;
END_ORGANIZATION_BLOCK

SYMBOL_TABLE
"EventsToPIC_DB"	DB 470	FB 470
"SSA_LOG_Value_Queue"	DB 1005	DB 1005	// PC Interface to log
"DB Prozesszeit"	DB 1010	DB 1010
"GCS7_E_ValveControl4Pos"	FB 20	FB 20	// GCS7: Element valve control with 4 positions
"GCS7_LiftingDevice"	FB 85	FB 85	// de: Hubzug
"GCS7_TractionDrive"	FB 86	FB 86	// Traction drive  de: Fahrantrieb
"SSA_MH_EventsToPIC"	FB 470	FB 470
"SSA_FU_Siemens"	FB 1811	FB 1811	// Siemens FU Profibus Communication
"SSA_SEW_MOVIDRIVE"	FB 1812	FB 1812	// SEW MOVIDRIVE Frequency Inverter Profibus Communication
"SSA_SIEMENS_MICROMASTER"	FB 1813	FB 1813	// SIEMENS MICROMASTER Frequency Inverter Profibus Communication
"SSA_SIEMENS_SINAMICS"	FB 1814	FB 1814	// SIEMENS SINAMICS Frequency Inverter Profibus Communication
"SSA_DANFOSS_VLT5000"	FB 1815	FB 1815	// DANFOSS VLT5000 Frequency Inverter Profibus Communication
"SSA_ABB"	FB 1816	FB 1816	// ABB ACS800 Frequency Inverter Profibus Communication
"SSA_NORD"	FB 1817	FB 1817	// NORDAC Frequency Inverter Profibus Communication
"SSA_SEW_MOVITRAC"	FB 1818	FB 1818	// SEW MOVITRAC Frequency Inverter Profibus Communication
"SB_DT_DT"	FC 34	FC 34	//  Subract DT - DT
"SB_DT_TM"	FC 35	FC 35	// Subtract DT Time
"Standard_MC07"	FC 130	FC 130
"Test_Simuli"	FC 999	FC 999	// Simulation beim Test
"Act_Value_LogConvert"	FC 1045	FC 1045	// LOG: GCS7 message convert
"SSA_MH_LogEntry_ActValue"	FC 1046	FC 1046	// LOG: Message entry in queue
"SSA_MH_LogCtrl_ActValue"	FC 1047	FC 1047	// LOG: Call queue controller
"SSA_MH_Increment_counter"	FC 1048	FC 1048
"GCS7_SecCtrlMainMalting"	FC 1060	FC 1060	// GCS7: Section control main program Special Version Malting Plant
"GCS7_SecCtrlSubMalting"	FC 1061	FC 1061	// GCS7: Section control subroutines Special Version Malting Plant
"Takt/Pause"	FC 1105	FC 1105
"Takt mit Pause"	FC 1106	FC 1106	// Takt/Pause AWR
"DPRD_DAT"	SFC 14	SFC 14	// Read Consistent Data of a Standard DP Slave
"DPWR_DAT"	SFC 15	SFC 15	// Write Consistent Data to a Standard DP Slave
"BLKMOV"	SFC 20	SFC 20	// Copy Variables
"SSA_MH_ProcessTime"	UDT 2000	UDT 2000	// Malthouse Actual time Process
"SSA_MH_StepTime"	UDT 2001	UDT 2001	// Malthouse Actual time Step
"SSA_MH_JobHeader"	UDT 2003	UDT 2003	// Malthouse SecNom: Job_Header
"SSA_MH_SecNomStandPIC"	UDT 2004	UDT 2004	// Malthouse SecNom: Standard Command PC
"SSA_MH_Step_Loading"	UDT 2011	UDT 2011	// Malthouse Step Loading
"SSA_MH_Step_Unloading"	UDT 2012	UDT 2012	// Malthouse Step Unloading
"SSA_MH_Step_Clearing"	UDT 2013	UDT 2013	// Malthouse Step Clearing
"SSA_Steep_Cmd"	UDT 2100	UDT 2100	// Steeping Section: Commands
"SSA_Steep_Par"	UDT 2101	UDT 2101	// Steeping Section: Parameter
"SSA_Steep_Recipe"	UDT 2102	UDT 2102	// Steeping Section: Recipe
"SSA_Steep_Analog"	UDT 2103	UDT 2103	// Steeping Section: Analog Values
"SSA_Steep_Recipe_Header"	UDT 2104	UDT 2104	// Steeping Section: Recipe Header
"SSA_Steep_Step"	UDT 2105	UDT 2105	// Steeping Section : Single Step
"SSA_Steep_Sum"	UDT 2106	UDT 2106	// Summary values for Steeping with sequencial conical steep
"SSA_Germ_Cmd"	UDT 2200	UDT 2200	// Germination Section: Commands
"SSA_Germ_Par"	UDT 2201	UDT 2201	// Germination Section: Parameter
"SSA_Germ_Recipe"	UDT 2202	UDT 2202	// Germination Section: Recipe
"SSA_Germ_Analog"	UDT 2203	UDT 2203	// Germination Section: Analog Values
"SSA_Germ_Recipe_Header"	UDT 2204	UDT 2204	// Germination Section:  Recipe Header
"SSA_Germ_Step"	UDT 2205	UDT 2205	// Germination Section: Single Step
"SSA_Kiln_Cmd"	UDT 2300	UDT 2300	// Kilning Section: Commands
"SSA_Kiln_Par"	UDT 2301	UDT 2301	// Kilning Section: Parameter
"SSA_Kiln_Recipe"	UDT 2302	UDT 2302	// Kilning Section: Recipe
"SSA_Kiln_Analog"	UDT 2303	UDT 2303	// Kilning Section: Analog Values
"SSA_Kiln_Recipe_Header"	UDT 2304	UDT 2304	// Kilning Section:  Recipe Header
"SSA_Kiln_Step"	UDT 2305	UDT 2305	// Kilning Section: Single Step
"CMDs_ILO_Funktion"	UDT 8015	UDT 8015	// Command and setpoints for one ILO-funktion
"SSA_LOG_Value"	UDT 10005	UDT 10005
END_SYMBOL_TABLE

TYPE "SSA_MH_ProcessTime"	// UDT 2000
VERSION : 0.1
  STRUCT
   Day : INT ;
   Hour : INT ;
   Min : INT ;
   Spare_93 : INT ;
   ProcessTimeActive : BYTE ;
   Spare_95 : BYTE ;
  END_STRUCT ;	
END_TYPE

TYPE "SSA_MH_StepTime"	// UDT 2001
VERSION : 0.1
  STRUCT
   SteptimeActHour : INT ;
   SteptimeActMin : INT ;
   SteptimeActMinOverall : INT ;
   StepTimeActHourTotal : INT ;
   Spare_85 : INT ;
  END_STRUCT ;	
END_TYPE

TYPE "SSA_MH_JobHeader"	// UDT 2003
VERSION : 0.1
  STRUCT
   StartSteepingProcess : DATE_AND_TIME ;
   Ident_of_Barley : DINT ;	//Ident (Code) of Barley
   Ident_of_Malt : DINT ;	//Ident (Code) of Malt
   Ident_Recipe_Steep_1 : DINT ;	//Ident (Code) of Steeping recipe first Steep
   Steeping_vessel_1 : INT ;	//Ident (Code) of Steeping Vessel first Steep (1 or 2)
   Ident_Recipe_Steep_2 : DINT ;	//Ident (Code) of Steeping recipe second Steep
   Steeping_vessel_2 : INT ;	//Ident (Code) of Steeping Vessel second Steep (1 or 2)
   Ident_Recipe_Germ : DINT ;	//Ident (Code) of Germinating recipe
   Germinating_vessel : INT ;	//Ident (Code) of Germinating Vessel
   Ident_Recipe_Kiln_1 : DINT ;	//Ident (Code) of Kilning recipe first Kiln
   Kilning_vessel_1 : INT ;	//Ident (Code) of Kilning Vessel first Kiln
   Ident_Recipe_Kiln_2 : DINT ;	//Ident (Code) of Kilning recipe second Kiln
   Kilning_vessel_2 : INT ;	//Ident (Code) of Kilning Vessel second Kiln
   Reserve001 : INT ;
   Reserve002 : INT ;
  END_STRUCT ;	
END_TYPE

TYPE "SSA_MH_SecNomStandPIC"	// UDT 2004
VERSION : 0.1
  STRUCT
   Par1On : STRUCT 	//Job parameters
    Cmd08 : BOOL ;	//Not used
    Cmd09 : BOOL ;	//Not used
    Cmd10 : BOOL ;	//Not used
    Cmd11 : BOOL ;	//Not used
    Cmd12 : BOOL ;	//Not used
    Cmd13 : BOOL ;	//Not used
    Cmd14 : BOOL ;	//Not used
    Cmd15 : BOOL ;	//Not used
    Cmd00 : BOOL ;	//Not used
    Cmd01 : BOOL ;	//Not used
    Cmd02 : BOOL ;	//Not used
    Cmd03 : BOOL ;	//Not used
    Cmd04 : BOOL ;	//Not used
    Cmd05 : BOOL ;	//Not used
    Cmd06 : BOOL ;	//Not used
    Cmd07 : BOOL ;	//Not used
   END_STRUCT ;
   Par2On : STRUCT 	//Job parameters
    Cmd08 : BOOL ;	//Not used
    Cmd09 : BOOL ;	//Not used
    Cmd10 : BOOL ;	//Not used
    Cmd11 : BOOL ;	//Not used
    Cmd12 : BOOL ;	//Not used
    Cmd13 : BOOL ;	//Not used
    Cmd14 : BOOL ;	//Not used
    Cmd15 : BOOL ;	//Not used
    Cmd00 : BOOL ;	//Not used
    Cmd01 : BOOL ;	//Not used
    Cmd02 : BOOL ;	//Not used
    Cmd03 : BOOL ;	//Not used
    Cmd04 : BOOL ;	//Not used
    Cmd05 : BOOL ;	//Not used
    Cmd06 : BOOL ;	//Not used
    Cmd07 : BOOL ;	//Not used
   END_STRUCT ;
   Par3On : STRUCT 	//Job parameters
    Cmd08 : BOOL ;	//Not used
    Cmd09 : BOOL ;	//Not used
    Cmd10 : BOOL ;	//Not used
    Cmd11 : BOOL ;	//Not used
    Cmd12 : BOOL ;	//Not used
    Cmd13 : BOOL ;	//Not used
    Cmd14 : BOOL ;	//Not used
    Cmd15 : BOOL ;	//Not used
    Cmd00 : BOOL ;	//Not used
    Cmd01 : BOOL ;	//Not used
    Cmd02 : BOOL ;	//Not used
    Cmd03 : BOOL ;	//Not used
    Cmd04 : BOOL ;	//Not used
    Cmd05 : BOOL ;	//Not used
    Cmd06 : BOOL ;	//Not used
    Cmd07 : BOOL ;	//Not used
   END_STRUCT ;
   Par4On : STRUCT 	//Job parameters
    Cmd08 : BOOL ;	//Not used
    Cmd09 : BOOL ;	//Not used
    Cmd10 : BOOL ;	//Not used
    Cmd11 : BOOL ;	//Not used
    Cmd12 : BOOL ;	//Not used
    Cmd13 : BOOL ;	//Not used
    Cmd14 : BOOL ;	//Not used
    Cmd15 : BOOL ;	//Not used
    Cmd00 : BOOL ;	//Not used
    Cmd01 : BOOL ;	//Not used
    Cmd02 : BOOL ;	//Not used
    Cmd03 : BOOL ;	//Not used
    Cmd04 : BOOL ;	//Not used
    Cmd05 : BOOL ;	//Not used
    Cmd06 : BOOL ;	//Not used
    Cmd07 : BOOL ;	//Not used
   END_STRUCT ;
   NotUsed01 : INT ;	//Not used
   NotUsed02 : INT ;	//Not used
   NotUsed03 : INT ;	//Not used
   NotUsed04 : INT ;	//Not used
   NotUsed05 : INT ;	//Not used
   NotUsed06 : INT ;	//Not used
   NotUsed07 : INT ;	//Not used
   NotUsed08 : INT ;	//Not used
   NotUsed09 : INT ;	//Not used
   NotUsed10 : INT ;	//Not used
   NotUsed11 : INT ;	//Not used
   NotUsed12 : INT ;	//Not used
   NotUsed13 : INT ;	//Not used
   NotUsed14 : INT ;	//Not used
   NotUsed15 : INT ;	//Not used
   NotUsed16 : INT ;	//Not used
  END_STRUCT ;	
END_TYPE

TYPE "SSA_MH_Step_Loading"	// UDT 2011
VERSION : 0.1
  STRUCT
   LoadingSpeed_1 : INT ;	//Speed round 1
   LoadingSpeed_2 : INT ;	//Speed round 2
   LoadingSpeed_3 : INT ;	//Speed round 3
   WaterPrefillingActivate : BYTE ;	//Activate WaterPrefilling
   sapre : BYTE ;
   TemperaturWater : DINT ;	//Setpoint watertemperature in °C (GMC)
   WaterPrefilling : DINT ;	//Water prefilling before grain input (m³) (UAN)
   Cooling : BYTE ;	//Activate Cooling System y/n (1/0) (GMC)
   GrainFillWithWater : BYTE ;	//0=no water fillling (grain intake only with anti-dust-spraying) (UAN)
   BankingLoadingScrew : INT ;	//Banking loading screw in mm
   LoadingLevelRound_1 : INT ;	//Level of Barley in first loading Round in mm
   LoadingLevelRound_2 : INT ;	//Level of Barley in second loading Round in mm
   LoadingLevelRound_3 : INT ;	//Level of Barley in third loading Round in mm
   OffsetLevelNextRound : INT ;	//Offset level of Barley in all next loading Rounds in mm
   LiftingPositionRound_1 : INT ;	//Lifting position in loading Round 1
   LiftingPositionRound_2 : INT ;	//Lifting position in loading Round 2
   LiftingPositionRound_3 : INT ;	//Lifting position in loading Round 3
   LiftingPositionRound_4 : INT ;	//Lifting position in loading Round 4
   LiftingPositionRound_5 : INT ;	//Lifting position in loading Round 5
   LiftingPositionRound_6 : INT ;	//Lifting position in loading Round 6
  END_STRUCT ;	
END_TYPE

TYPE "SSA_MH_Step_Unloading"	// UDT 2012
VERSION : 0.1
  STRUCT
   UnLoadingSpeed_1 : INT ;	//Speed round 0
   UnLoadingSpeed_2 : INT ;	//Speed round 1
   UnLoadingSpeed_3 : INT ;	//Speed round 2
   SPARE_INT0000 : INT ;	//Speed spare
   SPARE_INT0001 : INT ;	//Speed spare
   SPARE_INT0002 : INT ;	//Speed spare
   SPARE_DINT000 : DINT ;
   SPARE_DINT001 : DINT ;
   NextStep : INT ;	//Spare
   UnLoadingLevelRound_1 : INT ;	//Level of Greenmalt in first unloading Round in mm
   UnLoadingLevelRound_2 : INT ;	//Level of Greenmalt in second unloading Round in mm
   UnLoadingLevelRound_3 : INT ;	//Level of Greenmalt in third unloading Round in mm
   OffsetLevelNextRound : INT ;	//Spare
   SPARE_INT003 : INT ;
   SPARE_INT004 : INT ;
   StartUnloadAuto : BYTE ;	//Start unload automatically y/n (1/0)
   UnloadingWaterWithPump : BYTE ;	//Unloading water with pump y/n (1/0)
   SPARE_BYTE001 : BYTE ;
   SPARE_BYTE002 : BYTE ;
   SPARE_BYTE003 : BYTE ;
   SPARE_BYTE004 : BYTE ;
  END_STRUCT ;	
END_TYPE

TYPE "SSA_MH_Step_Clearing"	// UDT 2013
VERSION : 0.1
  STRUCT
   CleaningWater : DINT ;	//Volume of cleaning water in m³
   SPARE_DINT000 : DINT ;
   CleaningSpeed_1 : INT ;	//Speed round 0
   CleaningSpeed_2 : INT ;	//Speed round 1
   CleaningSpeed_3 : INT ;	//Speed round 2
   SPARE_INT0000 : INT ;	//Speed spare
   SPARE_INT0001 : INT ;	//Speed spare
   SPARE_INT0002 : INT ;	//Speed spare
   CoverCleaning_1 : BYTE ;	//Cover cleaning nozzle round 0 y/n (1/0) (GMC)
   CoverCleaning_2 : BYTE ;	//Cover cleaning nozzle round 1 y/n (1/0) (GMC)
   CoverCleaning_3 : BYTE ;	//Cover cleaning nozzle round 2 y/n (1/0) (GMC)
   Cleaning_1 : BYTE ;	//Cleaning nozzle 1
   Cleaning_2 : BYTE ;	//Cleaning nozzle 2
   SPARE_BYTE000 : BYTE ;
   CleaningLevel_1 : INT ;	//Wall cleaning level 1 in mm
   CleaningLevel_2 : INT ;	//Wall cleaning level 2 in mm
   CleaningLevel_3 : INT ;	//Wall cleaning level 3 in mm
   CleaningRounds : INT ;	//Number of Rounds
   StartCleaningAerNozzles : INT ;	//Starttime cleaning aeriation nozzles in min counted from start steptime
   TimeCleaningAerNozzles : INT ;	//Time cleaning aeriation nozzles in min
   TimeCleaningWall : INT ;	//Time cleaning wall in min
  END_STRUCT ;	
END_TYPE

TYPE "SSA_Steep_Cmd"	// UDT 2100
VERSION : 0.1
  STRUCT
   Functions : STRUCT
    StartLoading : BOOL ;	//Start Function Loading
    BreakLoading : BOOL ;	//Break Function Loading
    ContinueLoading : BOOL ;	//Continue Function Loading
    StopLoading : BOOL ;	//Stop Function Loading
    UnloadingManuel : BOOL ;	//Unloading in Manuel Mode, only for Kiln
    StartUnloading : BOOL ;	//Start Function Unloading
    BreakUnloading : BOOL ;	//Break Function Unloading
    ContinueUnloading : BOOL ;	//Continue Function Unloading
    StopUnloading : BOOL ;	//Stop Function Unloading
    StartCleaning : BOOL ;	//Start Function Cleaning
    BreakCleaning : BOOL ;	//Break Function Cleaning
    ContinueCleaning : BOOL ;	//Continue Function Cleaning
    CleaningReady : BOOL ;	//Stop Function Cleaning
    StartProcess : BOOL ;	//Comand of Future
    Comand16 : BOOL ;
    Comand17 : BOOL ;
   END_STRUCT ;
   General : STRUCT
    LiftingDeviceUP : BOOL ;	//Lifting device UP
    LiftingDeviceDOWN : BOOL ;	//Lifting device DOWN
    LiftingDeviceSTOP : BOOL ;	//Lifting device STOP
    LiftingDeviceRESET : BOOL ;	//Lifting device RESET FAULT
    LoadUnloadScrewINSIDE : BOOL ;	//Loading-Unloading Screw INSIDE (LEFT)
    LoadUnloadScrewOUTSIDE : BOOL ;	//Loading-Unloading Screw OUTSIDE (RIGHT)
    LoadUnloadScrewSTOP : BOOL ;	//Loading-UnloadingScrew STOP
    LoadUnloadScrewRESET : BOOL ;	//Loading-UnloadingScrew RESET FAULT
    DischargeFlapOPEN : BOOL ;	//Discharge flap OPEN
    DischargeFlapCLOSE : BOOL ;	//Discharge flap CLOSE
    DischargeFlapRESET : BOOL ;	//Discharge flap RESET FAULT
    RotatingFloorDrivesRIGHT : BOOL ;	//Rotating Floor Drives RIGHT
    RotatingFloorDrivesLEFT : BOOL ;	//Rotating Floor Drives LEFT
    RotatingFloorDrivesSTOP : BOOL ;	//Rotating Floor Drives STOP
    RotatingFloorDrivesRESET : BOOL ;	//Rotating Floor Drives RESET FAULT
    spare_16 : BOOL ;
   END_STRUCT ;
   SPARE0 : BYTE ;
   SPARE1 : BYTE ;
   SPARE2 : BYTE ;
   SPARE3 : BYTE ;
   SPARE4 : BYTE ;
   SPARE5 : BYTE ;
  END_STRUCT ;	
END_TYPE

TYPE "SSA_Steep_Par"	// UDT 2101
VERSION : 0.1
  STRUCT
   Switches1 : STRUCT
    StaOn24 : BOOL ;	//Example for comment: StaOn24WaterPumpA
    StaOn25 : BOOL ;
    StaOn26 : BOOL ;
    StaOn27 : BOOL ;
    StaOn28 : BOOL ;
    StaOn29 : BOOL ;
    StaOn30 : BOOL ;
    StaOn31 : BOOL ;
    PresetPump1 : BOOL ;
    PresetPump2 : BOOL ;
    PresetPump4 : BOOL ;
    PresetPump5 : BOOL ;
    PresetPump10 : BOOL ;
    PresetPump11 : BOOL ;
    a2 : BOOL ;
    a1 : BOOL ;
    FillWaterToMixingTank : BOOL ;
    FillBarleyToMixingTank : BOOL ;
    EmptyMixingTank : BOOL ;
    CleanMixingTank : BOOL ;
    StaOn12 : BOOL ;
    StaOn13 : BOOL ;
    StartWaterTransport : BOOL ;	//Start transport barley with pump P10/P11
    RestartWaterTransport : BOOL ;	//Restart transport barley from mixing tank to steep after blockage
    LiftingPositionRound_1 : BOOL ;
    LiftingPositionRound_2 : BOOL ;
    LiftingPositionRound_3 : BOOL ;
    LiftingPositionRound_4 : BOOL ;
    LiftingPositionRound_5 : BOOL ;
    LiftingPositionRound_6 : BOOL ;
    StaOn06 : BOOL ;
    StaOn07 : BOOL ;
   END_STRUCT ;
   Switches2 : STRUCT
    AutoLoading : BOOL ;
    StaOn25 : BOOL ;
    StaOn26 : BOOL ;
    StaOn27 : BOOL ;
    StaOn28 : BOOL ;
    StaOn29 : BOOL ;
    StaOn30 : BOOL ;
    StaOn31 : BOOL ;
    GMCFreshWaterSupplyOK : BOOL ;
    GMCBarleySlideOpen : BOOL ;
    StaOn18 : BOOL ;
    StaOn19 : BOOL ;
    StaOn20 : BOOL ;
    StaOn21 : BOOL ;
    StaOn22 : BOOL ;
    StaOn23 : BOOL ;
    StaOn08 : BOOL ;
    StaOn09 : BOOL ;
    StaOn10 : BOOL ;
    StaOn11 : BOOL ;
    StaOn12 : BOOL ;
    StaOn13 : BOOL ;
    StaOn14 : BOOL ;
    StaOn15 : BOOL ;
    StaOn00 : BOOL ;
    StaOn01 : BOOL ;
    StaOn02 : BOOL ;
    StaOn03 : BOOL ;
    StaOn04 : BOOL ;
    StaOn05 : BOOL ;
    StaOn06 : BOOL ;
    StaOn07 : BOOL ;
   END_STRUCT ;
   Values1 : STRUCT 	//Lineparameter data written by Host-System
    Value01 : DINT ;	//Example for comment: TurnoverTime [xxxs]
    TargetWeightFreshWater : DINT ;	//Setpoint fresh water in kg per Steep
    TargetWeightRecyclWater : DINT ;	//Setpoint recipe in 100 l per Steep
    TargetWeightOverflWater : DINT ;	//Setpoint overflow water in kg per Steep
    TimeCleanSurface : DINT ;	//Maximum Time to Clean Surface
    Value06 : DINT ;
    Value07 : DINT ;
    Value08 : DINT ;
    Value09 : DINT ;
    Value10 : DINT ;
    Value11 : DINT ;
    Value12 : DINT ;
    Value13 : DINT ;
    Value14 : DINT ;
    Value15 : DINT ;
    Value16 : DINT ;
    Value17 : DINT ;
    Value18 : DINT ;
    Value19 : DINT ;
    Value20 : DINT ;
    WeightSurname_1 : DINT ;	//weight surname after 1. steep in [kg]
    WeightSurname_2 : DINT ;	//weight surname after 2. steep in [kg]
    WeightSurname_3 : DINT ;	//weight surname after 3. steep in [kg]
    Value24 : DINT ;
    Value25 : DINT ;
    Value26 : DINT ;
    Value27 : DINT ;
    Value28 : DINT ;
    Value29 : DINT ;
    Value30 : DINT ;
   END_STRUCT ;
   FlagSec : STRUCT
    InfSameJobPrevSec : BOOL ;	//InfSameJobPrevSec von Section 1
    InfSameJobPrevSec_FN : BOOL ;	//InfSameJobPrevSec negative Flanke von Section 1
    InitVesselWeight : BOOL ;	//Initialisation of Vessel Weight
    Flag003 : BOOL ;
    CleanSurfaceTimer : BOOL ;	//Timer for Cleaning Surface
    CleanSurfaceIniFP : BOOL ;	//Initialisation Time to Clean Surface FP
    CleanSurfaceIni : BOOL ;	//Initialisation Time to Clean Surface
    Flag007 : BOOL ;
    FPStartLoading : BOOL ;
    ScanStartLoading : BOOL ;
    Flag0010 : BOOL ;
    FPStartFillWaterMixBin : BOOL ;
    ScanStartFillWaterMixBin : BOOL ;
    Flag0013 : BOOL ;
    FPStartFillBarleyMixBin : BOOL ;
    ScanStartFillBarleMixBin : BOOL ;
    DelayEmtyMIxBin : BOOL ;
    FPStartEmptyMixBin : BOOL ;
    ScanStartEmptyMixBin : BOOL ;
    Flag0019 : BOOL ;
    FPStartCleanMixBin : BOOL ;
    ScanStartCleanMixBin : BOOL ;
    Flag0022 : BOOL ;
    FPStartUnLoading : BOOL ;
    ScanStartUnLoading : BOOL ;
    Flag0025 : BOOL ;
    EmptyPipes : BOOL ;
    PipesEmptied : BOOL ;
    Flag0028 : BOOL ;
    TimeCleaningWallLoad : BOOL ;
    TimeCleaningWallEdge : BOOL ;
    FaultDB_Copy : BOOL ;	//Fault DB Copy FC49
   END_STRUCT ;
   FlagGen : STRUCT
    WindAlarm : BOOL ;	//Wind speed is too high
    TurningStarted : BOOL ;	//Germination turning is started
    WetStep : BOOL ;	//Active Step is Wet Step
    Flag003 : BOOL ;
    SteepFilledWithSorghum : BOOL ;	//Steep is filled with sorghum
    Flag005 : BOOL ;
    Flag006 : BOOL ;
    Flag007 : BOOL ;
    LOAD_VAL_HUB1 : BOOL ;	//Counter lifting device 1
    LOAD_VAL_HUB2 : BOOL ;	//Counter lifting device 2
    LOAD_VAL_DRIVE : BOOL ;	//Counter driving device
    LOAD_VAL_AFTER_FAILURE : BOOL ;	//Counter saved datas after failure
    Flag0012 : BOOL ;
    Flag0013 : BOOL ;
    OverflowWaterReached : BOOL ;	//Overflow water volume is reached
    SteepFull : BOOL ;	//Steep is full
    InterlockedFunktionMode : BOOL ;
    ILO_CmdResetFault : BOOL ;
    Flag0018 : BOOL ;
    Flag0019 : BOOL ;
    Flag0020 : BOOL ;
    Flag0021 : BOOL ;
    Flag0022 : BOOL ;
    Flag0023 : BOOL ;
    Flag0024 : BOOL ;
    Flag0025 : BOOL ;
    Flag0026 : BOOL ;
    Flag0027 : BOOL ;
    Flag0028 : BOOL ;
    Flag0029 : BOOL ;
    Flag0030 : BOOL ;
    Flag0031 : BOOL ;
   END_STRUCT ;
   Spare136 : ARRAY  [136 .. 139 ] OF BYTE ;
   ParIntProcess : STRUCT 	//Processparameter data
    UnloadungRounds : INT  := 2;
    LoadungRounds : INT  := 2;	//
    LoadingOverlap : INT  := 10;	//overlap in ° by loading
    UnloadingOverlap : INT  := 20;	//overlap in ° by unloading
    TurningLevelMeasure : INT  := 5;	//Turning in ° by level measure
    DiffLevelMeasure : INT  := 3;	//Max. Difference in mm by level measure
    DownLevelPerPulse : INT ;
    Value8 : INT ;
    ActualTimeSpraying : INT ;
    ActualDelaySpraying : INT ;
    Value11 : INT ;
    Value12 : INT ;
    ActualTimeCirculation : INT ;
    ActualPauseCirculation : INT ;
    Value15 : INT ;
    ActualTimeAeriation : INT ;
    ActualPauseAeriation : INT ;
    ActualDelayAeriation : INT ;
    Value19 : INT ;
    SetpointDrainTimeACS : INT ;
    ActTimeDrainAftCleanSurf : INT ;
    StateWordSteep : INT ;	//State-Number of the active Step
    TimeBalanceWater : INT ;	//time to balance water levels between steeps in [min]
    Value24 : INT ;
    Value25 : INT ;
    TargetOverflowTimeSteep : INT ;	//Abschwemmzeit pro Konusweiche in sec
    StartTimeInterval_3 : INT ;	//Startzeit 3.Interwall in sec
    StartTimeInterval_2 : INT ;	//Startzeit 2.Interwall in sec
    ActOverflowTimeSteep : INT ;	//Laufzeit Gesamt-Interwall pro Konusweiche in sec
    TarPos_ILO_LiftDev : INT ;	//Target positon lifting devices from ILO-Mode
    TarPos_ILO_FreshAir : INT ;	//Target positon fresh air flap from ILO-Mode
    TarPos_ILO_ExhaustAir : INT ;	//Target positon exhaust air flap from ILO-Mode
    Speed_ILO_Fan : INT ;	//Target speed germinatimng fan from ILO-Mode
    Speed_ILO_TravelDrive : INT ;	//Target speed travelling drive from ILO-Mode
    TargetTemperature_ILO : INT ;	//Target temperature from ILO-Mode
    ActTimeCleanMixTank : INT ;
    TarPos_ILO_WasteAir : INT ;
    Value38 : INT ;
    Value39 : INT ;
    SetpointBackwaterFlap060 : INT ;
    SetpointBackwaterFlap160 : INT ;
    SetpointTimeCleanMixTank : INT ;
    Value43 : INT ;
    Value44 : INT ;
    Value45 : INT ;
    Value46 : INT ;
    Value47 : INT ;
    Value48 : INT ;
    Value49 : INT ;
    ActualStep : INT ;	//Actual Step for visu
   END_STRUCT ;
   ParIntMachine : STRUCT 	//Machine parameter data
    ActualStep : INT ;	//Actual process step
    MAX_HUB_DIFF : INT  := 36;	//Max. Hubdifferenz zwischen Hubzug 1 + 2
    REINIGUNGSHOEHE : INT  := 100;	//Reinigungshoehe in mm
    MAX_SCHIEFLAGE : INT  := 150;	//Max. Schieflage zwischen Hubzug 1 + 2
    IMPULSE_HUBZUG1_OBEN : INT  := 480;	//Impulse : Hubantrieb 1 normieren bei Endpos.oben
    IMPULSE_HUBZUG2_OBEN : INT  := 480;	//Impulse : Hubantrieb 2 normieren bei Endpos.oben
    POSITION_HUBZUG1_OBEN : INT  := 1055;	//Hoehe in mm
    POSITION_HUBZUG2_OBEN : INT  := 1055;	//Hoehe in mm
    IMPULSE_RUNDE : INT  := 816;	//Impulse : Fahrantriebantrieb eine Runde (Diesen Wert bei der IBS ermitteln!!)
    SollwertFahrantrWenden : WORD  := W#16#DEF;	//21,7% von 100 Hz
    LiftDevMinPos : INT  := 100;	//Lifting device minimal position for rotation backwards
    FUELLHOEHE_PRODUKT : INT ;	//Produkt-Füllhöhe
    SOLLWERT_HUBZUG1_HOEHE : INT ;
    Value14 : INT ;
    Value15 : INT ;
    LoadingLevelRound_4 : INT ;	//Calculated value level in 4. round
    LoadingLevelRound_5 : INT ;	//Calculated value level in 5. round
    LoadingLevelRound_6 : INT ;	//Calculated value level in 6. round
    LiftingPositionRound_4 : INT ;	//Calculated value lifting position in loading round 4
    LiftingPositionRound_5 : INT ;	//Calculated value lifting position in loading round 5
    LiftingPositionRound_6 : INT ;	//Calculated value lifting position in loading round 6
    Value22 : INT ;
    Value23 : INT ;
    DelayEmptyMixTank : INT ;
    Value25 : INT ;
    Value26 : INT ;
    Value27 : INT ;
    Value28 : INT ;
    Value29 : INT ;
    Value30 : INT ;
    SteepingBoxNumber : INT ;
    Value32 : INT ;
    Value33 : INT ;
    Value34 : INT ;
    Value35 : INT ;
    Value36 : INT ;
    Value37 : INT ;
    Value38 : INT ;
    Value39 : INT ;
    Value40 : INT ;
    Value41 : INT ;
    Value42 : INT ;
    Value43 : INT ;
    Value44 : INT ;
    Value45 : INT ;
    Value46 : INT ;
    Value47 : INT ;
    Value48 : INT ;
    Value49 : INT ;
    LastWetsteep : INT ;	//Parameter "DelayNextAeriationCycle" from last wetsteep
   END_STRUCT ;
   FlagFunction_0 : STRUCT 	//Flags section
    AeriationConeSelected : BOOL ;	//Example for comment: Inf24WaterPumpA
    AeriationConeActive : BOOL ;
    AeriationHTubeSelected : BOOL ;
    AeriationHTubeActive : BOOL ;
    FNFirstAerHTFinished : BOOL ;
    FirstAerHTFinished : BOOL ;
    CleaningSurfaceFinished : BOOL ;
    StoreAerDuringWaterFill : BOOL ;
    ImpulsAbraeumenGestartet : BOOL ;
    AbraeumenGestartetFP : BOOL ;
    AbraeumenGestartet : BOOL ;
    AutostartAbraeumenFP : BOOL ;
    AutostartAbraeumen : BOOL ;
    MerkerBeladenGestartet : BOOL ;
    MerkerEntladenGestartet : BOOL ;
    MerkerBeladenGestartetFP : BOOL ;
    ImpulsBeladenGestartet : BOOL ;
    MerkerEntladGestartetFP : BOOL ;
    ImpulsEntladenGestartet : BOOL ;
    FlagCleaningStartedFP : BOOL ;
    ImpulseCleaningStarted : BOOL ;
    CleaningGestartet : BOOL ;
    ImpulsMeasureHightLevel : BOOL ;
    MeasureHightLevelFN : BOOL ;
    FlagSprayingStartingFP : BOOL ;
    SprayingStarting : BOOL ;
    Inf02 : BOOL ;
    CleaningPipesAndFloor : BOOL ;
    CleanPipesAndFloorActive : BOOL ;
    CleanPipesAndFloorReady : BOOL ;
    InfReleaseUnloading : BOOL ;
    ErrorLevelMeasure : BOOL ;
   END_STRUCT ;
   FlagMachine : STRUCT 	//flags machine funktion
    Hubzug1_Low : BOOL ;	//Hubzug 1 Richtungsvorwahl senken
    Hubzug1_High : BOOL ;	//Hubzug 1 Richtungsvorwahl heben
    Hubzug2_Low : BOOL ;	//Hubzug 2 Richtungsvorwahl senken
    Hubzug2_High : BOOL ;	//Hubzug 2 Richtungsvorwahl heben
    Stop_Hubzuege : BOOL ;	//Differenz Hub1-Hub2>Vorgabewert
    Hubzug1_Speed_Ctr : BOOL ;	//Hubantrieb 1 innen Drehueberwachung
    Hubzug2_Speed_Ctr : BOOL ;	//Hubantrieb 2 aussen Drehueberwachung
    Produktsensor_Ctr : BOOL ;	//Produktsensor-Ueberwachung
    Hubzug1_Stop_NullPos_man : BOOL ;	//Hoehe Hubzug 1 <= NULL-Position
    Hubzug2_Stop_NullPos_man : BOOL ;	//Hoehe Hubzug 2 <= NULL-Position
    Hubdiff1_2 : BOOL ;	//Hubdifferenz Hub1 > Hub2
    Hubdiff2_1 : BOOL ;	//Hubdifferenz Hub2 > Hub1
    Hubzug1_Hoch : BOOL ;	//Hubzug 1 Isthoehe > 300mm (Freigabe Ausraeumglocke schliessen) und Hubzuege heb
    Hubzug2_Hoch : BOOL ;	//Hubzug 2 Isthoehe > 300mm (Freigabe Ausraeumglocke schliessen) und Hubzuege heb
    Start_Hubzuege_Heben : BOOL ;	//Hubzuege heben
    Hubdiff1_2_NegAlt : BOOL ;	//Hubdifferenz Hub1 > Hub2 Alt-Signal
    Hubdiff1_2_NegFlag : BOOL ;	//Hubdifferenz Hub1 > Hub2 Flanken-Signal
    Hubdiff2_1_NegAlt : BOOL ;	//Hubdifferenz Hub2 > Hub1 Alt-Signal
    Hubdiff2_1_NegFlag : BOOL ;	//Hubdifferenz Hub2 > Hub1 Flanken-Signal
    Fahrantrieb_Speed_Ctr1 : BOOL ;	//Fahrantrieb Drehueberwachung
    Fahrantrieb_Start_ok : BOOL ;	//Es sind weniger als 2 Fahrantriebe nicht gestartet
    Fahrantrieb_FU_Fault : BOOL ;	//Sammelstörung von allen 12 FU's
    Fahrantriebe_Fwd_Rev : BOOL ;	//Aktuelle Drehrichtung Fahrantriebe (0=Fwd; 1=Rev)
    Fahrantriebe_Vorwaerts : BOOL ;	//Fahrantriebe Ausgang Richtung Vorwärts
    Fahrantriebe_Rueckwaerts : BOOL ;	//Fahrantriebe Ausgang Richtung Rückwärts
    NULL_INDEX_FP : BOOL ;
    ImpulsNullstellung : BOOL ;
    ImpulsNullstellungFP : BOOL ;
    WEGMESSUNG_0 : BOOL ;
    WEGMESSUNG_0_FLAG : BOOL ;
    Hubzug1_ueber_MinPos : BOOL ;	//Hubzug 1 mehr als 100mm ueber ihrer Nullposition
    Hubzug2_ueber_MinPos : BOOL ;	//Hubzug 2 mehr als 100mm ueber ihrer Nullposition
   END_STRUCT ;
   FlagFunction_1 : STRUCT 	//Flags functions
    StepLoading : BOOL ;	//Function Loading is active
    StepUnloading : BOOL ;	//Function Unloading is active
    StepCleaning : BOOL ;	//Function Cleaning is active
    LoadingBreak : BOOL ;	//Function Loading is interrupted
    UnloadingBreak : BOOL ;	//Function Unloading is interrupted
    CleaningBreak : BOOL ;	//Function Cleaning is interrupted
    FinishLoading : BOOL ;	//Function Loading is finished
    FinishUnloading : BOOL ;	//Function Unloading is finished
    FinishCleaning : BOOL ;	//Function Cleaning is finished
    TurningMeasure : BOOL ;	//Turning to measure hight level
    MeasureHightLevel : BOOL ;	//Measure hight level
    TurningZeroPoint : BOOL ;	//Turning to zero point
    Runde_1 : BOOL ;	//Fahrantrieb 1.Runde
    Runde_2 : BOOL ;	//Fahrantrieb 2.Runde
    Runde_3 : BOOL ;	//Fahrantrieb 3.Runde
    Runde_4 : BOOL ;	//Fahrantrieb 4.Runde
    Runde_5 : BOOL ;	//Fahrantrieb 5.Runde
    Runde_6 : BOOL ;	//Fahrantrieb 6.Runde
    Beladung_beendet : BOOL ;	//Fahrantrieb; Beladung_beendet
    Entladerunden_erreicht : BOOL ;	//Fahrantrieb; Entladerunden erreicht
    Reinigungsrunden_erreich : BOOL ;	//Fahrantrieb; Reinigungsrunden erreicht
    TurningStart : BOOL ;	//Start turning
    TurningStop : BOOL ;	//Stop turning
    TurningLeft : BOOL ;	//Germination turning left, with spraying
    TurningRight : BOOL ;	//Germination turning right, without spraying
    LoadFirstPartEnd : BOOL ;	//Grundschicht ist bedeckt, prozess kann starten
    TurningWithSpraying : BOOL ;	//Turning-round in this step with spraying
    TurningWithoutSpraying : BOOL ;	//Turning-round in this step without spraying
    UnloadEnd : BOOL ;	//Kilning box is unloaded
    UnloadSecondPartEnd : BOOL ;
    UnloadFirstPart : BOOL ;
    UnloadSecondPart : BOOL ;
   END_STRUCT ;
   FlagProcess : STRUCT 	//Flags process
    ProcessActive : BOOL ;	//Process is active
    ProcessStartFP : BOOL ;
    ProcessStartScan : BOOL ;
    ProcessEnd : BOOL ;
    ProcessEndFP : BOOL ;
    ProcessEndScan : BOOL ;
    NewStep : BOOL ;
    ReleaseProcessStart : BOOL ;
    FillingConditionatedWate : BOOL ;
    FillingFreshWater : BOOL ;
    SprayDuringFilling : BOOL ;
    AeriationDuringWaterFill : BOOL ;
    AeriatDurWaterFillFinish : BOOL ;	//
    SteepWaterFilled : BOOL ;	//
    SteepWaterFilledBySensor : BOOL ;	//
    CleaningSurface : BOOL ;
    RunningCyclicAeriation : BOOL ;
    AeriationActive : BOOL ;	//
    SprayDuringAeriation : BOOL ;	//
    FillingWaterFN : BOOL ;	//
    FillingFreshWaterFP : BOOL ;	//
    DrainWater : BOOL ;
    SteepWaterDrainedStopAer : BOOL ;
    SteepWaterDrainedStartCO : BOOL ;
    SprayingDuringCO2Suck : BOOL ;
    SprayDuringCO2SuckActive : BOOL ;
    CO2ExhaustDurUnloading : BOOL ;	//Exhaust CO2 during unloading
    CO2Exhaust : BOOL ;	//Exhaust CO2 during dry steep
    CO2SuckDurUnloading_3 : BOOL ;	//
    CO2SuckDurUnloading_4 : BOOL ;	//
    VentilatorDrehzahlMax : BOOL ;
    FP_SendResultToPIC : BOOL ;
   END_STRUCT ;
   FlagProcess1 : STRUCT 	//Flags process
    CirculationContinious : BOOL ;	//Proces is in stap droogcyclus 2,4,..enzv
    CirculationIntermitt : BOOL ;
    CoolingRequired : BOOL ;
    ErrorMech_NoNextStep : BOOL ;
    CirculIntermittActive : BOOL ;
    CirculIntermittPause : BOOL ;
    AeriationIntermittActive : BOOL ;
    AeriationIntermittPause : BOOL ;
    FP_WaterFill : BOOL ;
    HP_WaterFill : BOOL ;
    FPCleaningSurface : BOOL ;
    FillWaterForCleanSurf : BOOL ;
    WaterFilledForCleanSurf : BOOL ;
    DrainWaterAfterCleanSurf : BOOL ;
    WaterDrainedAfterClSurf : BOOL ;
    Cooling : BOOL ;	//Cooling ON
    HubzuegeUeberProdukt : BOOL ;
    UnloadLevelReachedFP : BOOL ;
    ImpulsUnloadLevelReached : BOOL ;
    Inf11 : BOOL ;
    AirHumifidication : BOOL ;
    Inf13 : BOOL ;
    WaterPreFillingDone : BOOL ;
    CmdAeriationActive : BOOL ;
    AeriationConeNozzle : BOOL ;
    AeriationHeinekenTube : BOOL ;
    NoAerationBySteepFull : BOOL ;	//No release aeration by cleaning surface
    SteepCleanSurfaceActive : BOOL ;	//Cleaning surface in steep running
    BalanceWaterLevels : BOOL ;	//Balance water levels between steeps
    BalanceWaterLevelsActive : BOOL ;	//Time to balance water levels running
    StepWetsteep : BOOL ;	//Odd stepnumber = wetsteep
    StepDrysteep : BOOL ;	//even stepnumber = drysteep
   END_STRUCT ;
   FlagGen33 : STRUCT 	//FlagProcess
    WaterStationOnline : BOOL ;	//PLC Water-Tanks is online
    SufficientlyCondWater : BOOL ;	//Sufficiently conditionated water in tanks
    SufficientlyFreshWater : BOOL ;	//Sufficiently fresh water in tanks
    Inf27 : BOOL ;
    Inf28 : BOOL ;
    Inf29 : BOOL ;
    Inf30 : BOOL ;
    Inf31 : BOOL ;
    WaterDrainReady : BOOL ;	//Water drain pumps and tank are ready
    Inf17 : BOOL ;
    Inf18 : BOOL ;
    Inf19 : BOOL ;
    FlagNewAeriatinCycle : BOOL ;
    Inf21 : BOOL ;
    Inf22 : BOOL ;
    Inf23 : BOOL ;
    Inf08 : BOOL ;
    Inf09 : BOOL ;
    Inf10 : BOOL ;
    Inf11 : BOOL ;
    Inf12 : BOOL ;
    Inf13 : BOOL ;
    Inf14 : BOOL ;
    Inf15 : BOOL ;
    Inf00 : BOOL ;
    Inf01 : BOOL ;
    Inf02 : BOOL ;
    Inf03 : BOOL ;
    Inf04 : BOOL ;
    Inf05 : BOOL ;
    Inf06 : BOOL ;
    ErrorCopy : BOOL ;
   END_STRUCT ;
   ProcessValue : STRUCT 	//Process values, used only in the PLC
    SetpointCondWater : DINT ;	//Setpoint from recipe
    ActualCondWater : DINT ;	//Actual value
    ActCondWaterVol_Saved : DINT ;	//Summary volume Conditioned water
    SetpointFreshWater : DINT ;	//Setpoint from recipe
    ActualFreshWater : DINT ;	//Actual value
    ActFreshWaterVol_Saved : DINT ;	//Summary volume Fresh water
    SetpointCleaningWater : DINT ;	//Setpoint from recipe
    ActualCleaningWater : DINT ;	//Actual value
    ActCleaninWaterVol_Saved : DINT ;	//Summary volume Cleaning water
    SummaryWaterOverall : DINT ;	//Summary volume water for checking waterflow
    MinWaterLevelAeriation : DINT ;	//Minimal water level for aeriation
    Profimess_Command : DINT ;	//command to read data from Profimess
    ActAeriationTime : INT ;	//old - ActAeriationPause
    NomAeriationPause : INT ;
    ActAeriationPause : INT ;
    ActTimeBalanceWater : INT ;	//Actual time to balance water levels between steeps in [min]
    ActTimeWaterDrain : INT ;
    RemainingDrainTime : INT ;
    ActSteptimeCleaning : INT ;
    ActSteptimeCleaningActiv : INT ;
    ProductLevel : INT ;
    SetpointUnloadLevel : INT ;
    ActualSpeedTravDrive : INT ;
    StepNrActCopy : INT ;
    StartStepAct : DATE_AND_TIME ;
    ActualTime : DATE_AND_TIME ;
    BreakPoint : DATE_AND_TIME ;
    StartCooling : DATE_AND_TIME ;
    StepTimeAct : TIME ;
    Value25 : TIME ;
    Value26 : TIME ;
    Value27 : TIME ;
   END_STRUCT ;
   Spare484 : ARRAY  [484 .. 499 ] OF BYTE ;
   ProcessValueReal : STRUCT 	//Process real values, used only in the PLC
    ReglerVentilator_Gain : REAL ;
    ReglerVentilator_I_Time : REAL ;
    Faktor_Um_Zuluftklappe_R : REAL ;	//Weg/Zeit-Faktor der Um- Zuluftklappe 1.1
    Faktor_AbluftSchwenkk1_R : REAL ;	//Weg/Zeit-Faktor derAbmluft-Schwenkklappe 1
    Faktor_AbluftSchwenkk2_R : REAL ;	//Weg/Zeit-Faktor derAbmluft-Schwenkklappe 2
    Fahrzeit_Um_Zuluftklap_R : REAL ;	//Fahrzeit der Um- Zuluftklappe 1.1
    Fahrzeit_AbluftSchwen1_R : REAL ;	//Fahrzeit der Abluft-Schwenkklappe 1
    Fahrzeit_AbluftSchwen2_R : REAL ;	//Fahrzeit der Abluft-Schwenkklappe 2
    Position_Um_Zuluftklap_R : REAL ;	//Position der Um- Zuluftklappe 1.1
    Position_AbluftSchwek1_R : REAL ;	//Position der Abluft-Schwenkklappe 1
    Position_AbluftSchwek2_R : REAL ;	//Position der Abluft-Schwenkklappe 2
    SollPos_Um_Zuluftklapp_R : REAL ;	//Soll-Position der Um- Zuluftklappe 1.1
    Value13 : REAL ;
    Value14 : REAL ;
    Value15 : REAL ;
    Value16 : REAL ;
    Value17 : REAL ;
    Value18 : REAL ;
    Value19 : REAL ;
    Value20 : REAL ;
    Value21 : REAL ;
    Value22 : REAL ;
    Value23 : REAL ;
    Value24 : REAL ;
    Profimess_Wirkleistung : REAL ;
    Profimess_Blindleistung : REAL ;
    Profimess_Frequenz : REAL ;
    Profimess_Wirkleist_Psec : REAL ;
    Profimess_Arbeit_Batch : REAL ;
    EnergieKWs : REAL ;
   END_STRUCT ;
   MachineValue : STRUCT 	//Machine values, used only in the PLC
    ISTWERT_FAHRANTRIEB_POSI : INT ;	//Ist-Position Fahrantrieb
    FAHRANTRIEB_UMDREHUNGEN : INT ;	//Rundenzaehler Fahrantrieb
    IST_HUB_DIFF : INT ;	//Istwert Hubdifferenz zwischen Hubzug 1 + 2
    ISTWERT_HUBZUG1_Z_IMP : INT ;	//Istwert Zaehlimpulse Hubzug 1
    ISTWERT_HUBZUG2_Z_IMP : INT ;	//Istwert Zaehlimpulse Hubzug 2
    SCHRAEGE_HUB1_HUB2 : INT ;	//Schraege Hub 1 > Hub 2
    SOLLWERT_HUBZUG1_HOEHE : INT ;
    SOLLWERT_HUBZUG2_HOEHE : INT ;
    ISTWERT_HUBZUG1_HOEHE : INT ;
    ISTWERT_HUBZUG2_HOEHE : INT ;
    SCHRAEGE_HUB1_MINUS_HUB2 : INT ;	//Schraege Hub 1 minus Hub 2
    SCHRAEGE_HUB2_MINUS_HUB1 : INT ;	//Schraege Hub 2 minus Hub 1
    BELADERUNDEN_START_HUB : INT ;	//Anhebeposition in Grad
    ISTWERT_FAHRANTRIE_Z_IMP : INT ;	//Istwert Zaehlimpulse Fahrantrieb
    Fahrantriebe_Gestartet : INT ;	//Zaehlwert der gestarteten Fahrantriebe
    SollwertFahrantrieb : WORD ;
    Fahrzeit_Reinigungswagen : INT ;	//Fahrzeit des Reinigungswagens unter der Horde
    Position_Reinigungswagen : INT ;	//Position der Reinigungswagens unter der Horde
    ISTWERT_HUBZUG1_DOPPEL : DINT ;	//Hubzug 1 : Hoehe [mm] Rechenwert
    ISTWERT_HUBZUG2_DOPPEL : DINT ;	//Hubzug 2 : Hoehe [mm] Rechenwert
    BELADERUNDEN_HUB_IMP : DINT ;	//Anhebeposition in Pulsen
    FAHR_GRAD_DOPPEL : DINT ;	//Fahrantrieb : Umdrehung in Grad Rechenwert
    Value14 : DINT ;
    Value15 : DINT ;
    FloorPositionPercent : DINT ;	//Floor position percentagewise
    CalcMinLvlWaterAeriation : DINT ;	//Calculated from Recipe m3 to l
    Value18 : DINT ;
    Value19 : DINT ;
    ActualWeightSteep : DINT ;	//Actual weight barley in steep
    ZeroWeightSteep : DINT ;	//Zero weight steep
    WeightSteepCO2Exhaust : DINT ;	//Minimal weight steep for CO2 exhaust
    SteepFullWeight : DINT ;	//Maximal weight full steep
    Value24 : DINT ;
    Value25 : DINT ;
    BarleyLevel : INT ;	//Barley level
    WaterLevel : INT ;	//Water level
    LAST_LOADING_LEVEL : INT ;	//Safe last loading level
    LAST_LIFTING_POSITION : INT ;	//Safe last lifting position
    HUBZUG1_Z_IMP_HOLD : DINT ;	//Istwert Zaehlimpulse Hubzug 1 gespeichert
    HUBZUG2_Z_IMP_HOLD : DINT ;	//Istwert Zaehlimpulse Hubzug 2 gespeichert
    FAHRANTRIEB_Z_IMP_HOLD : DINT ;	//Istwert Zaehlimpulse Fahrantrieb gespeichert
   END_STRUCT ;
   MachineValueReal : STRUCT 	//Machine real values, used only in the PLC
    HUB1_MM_PRO_IMPULS : REAL  := 2.197917e+000;	//Hubzug 1 : Hoehe [mm] pro Hubimpuls
    HUB2_MM_PRO_IMPULS : REAL  := 2.197917e+000;	//Hubzug 2 : Hoehe [mm] pro Hubimpuls
    FAHRANTRIEB_IMP_GRAD : REAL  := 4.411765e-001;	//Winkelgrad pro Fahrimpuls (wird automatisch berechnet)
    FAHR_GRAD_PRO_IMPULS : REAL ;	//Fahrantrieb : Umdrehung in Grad pro Fahrimpuls Real-Rechenwert
    IMPULSE_RUNDE_REAL : REAL ;	//Impulse : Fahrantrieb eine Runde Real-Rechenwert
    Faktor_Reinigungswagen_R : REAL ;	//Weg/Zeit-Faktor Reinigungswagens unter der Horde
    Fahrzeit_Reinigungswag_R : REAL ;	//Fahrzeit der Reinigungswagens unter der Horde
    Position_Reinigungswag_R : REAL ;	//Position der Reinigungswagens unter der Horde
    FAHRANTRIEB_IMP_PROZ : REAL ;	//Prozentzahl pro Fahrimpuls (wird automatisch berechnet)
    BELADERUNDEN_START_HUB : REAL ;	//Anhebeposition von % in Grad
    Value11 : REAL ;
    Value12 : REAL ;
    Value13 : REAL ;
    Value14 : REAL ;
    Value15 : REAL ;
    Value16 : REAL ;
    Value17 : REAL ;
    Value18 : REAL ;
    Value19 : REAL ;
    Value20 : REAL ;
    Value21 : REAL ;
    Value22 : REAL ;
    Value23 : REAL ;
    Value24 : REAL ;
    Value25 : REAL ;
    Value26 : REAL ;
    Value27 : REAL ;
    Value28 : REAL ;
    Value29 : REAL ;
    Value30 : REAL ;
   END_STRUCT ;
   Spare860 : INT ;
   Spare862 : INT ;
   Spare864 : INT ;
   Spare866 : INT ;
   Spare868 : INT ;
   Spare870 : INT ;
   Spare872 : INT ;
   Spare874 : INT ;
   Spare876 : INT ;
   Spare878 : INT ;
   Spare880 : INT ;
   Spare882 : INT ;
   Spare884 : INT ;
   Spare886 : INT ;
   Spare888 : INT ;
   Spare890 : INT ;
   Spare892 : INT ;
   Spare894 : INT ;
   Error : STRUCT
    Value : INT ;
    Bit : BOOL ;
   END_STRUCT ;
  END_STRUCT ;	
END_TYPE

TYPE "SSA_Steep_Recipe"	// UDT 2102
VERSION : 0.1
  STRUCT
   RecipeHeader : UDT 2104;
   Step : ARRAY  [1 .. 7 ] OF UDT 2105;
  END_STRUCT ;	
END_TYPE

TYPE "SSA_Steep_Analog"	// UDT 2103
VERSION : 0.1
  STRUCT
   NumberOfAeriationLines : INT ;	//Number of lines (valves) of Aeriation
   DelayNextValve : INT ;	//Delay to open next valve in sec
   DelayNextAeriationCycle : INT ;	//Delay between two Aeriation-Starts in min
   SpeedVentilator1 : INT ;	//Setpoint Fanspeed in % CO2 suck off Fan 1
   SpeedVentilator2 : INT ;	//Setpoint Fanspeed in % CO2 suck off Fan 2
   SpeedVentilator3 : INT ;	//Setpoint Fanspeed in % CO2 suck off Fan 3
   SpeedVentilator4 : INT ;	//Setpoint Fanspeed in % CO2 suck off Fan 4
   DrainTimeWaterAeriation : INT ;	//Time to drain Water before stop Aeriation in min
   DrainTimeWaterCO2Suck : INT ;	//Time to drain Water before Start CO2 suck off in min
   StartSpraying : INT ;	//Starttime spraying in min counted from start steptime
   TimeSpraying : INT ;	//Time one Round spraying
   DelaySpraying : INT ;	//Delay between two starts spraying
   Spare24 : INT ;
   Spare26 : INT ;
   Spare28 : INT ;
   Spare30 : INT ;
   Spare32 : INT ;
   Spare34 : INT ;
   Change : STRUCT
    SpeedVentilatorBasicGer : BOOL ;	//the analog value has change if there is a bit
    PositFreshAirFlapBasic : BOOL ;	//the analog value has change if there is a bit
    NumberOfAeriationLines : BOOL ;	//the analog value has change if there is a bit
    DelayNextValve : BOOL ;	//the analog value has change if there is a bit
    DelayNextAeriationCycle : BOOL ;	//the analog value has change if there is a bit
    SpeedVentilator1 : BOOL ;	//the analog value has change if there is a bit
    SpeedVentilator2 : BOOL ;	//the analog value has change if there is a bit
    SpeedVentilator3 : BOOL ;	//the analog value has change if there is a bit
    SpeedVentilator4 : BOOL ;	//the analog value has change if there is a bit
    DrainTimeWaterAeriation : BOOL ;	//the analog value has change if there is a bit
    DrainTimeWaterCO2Suck : BOOL ;	//the analog value has change if there is a bit
    StartSpraying : BOOL ;	//the analog value has change if there is a bit
    TimeSpraying : BOOL ;	//the analog value has change if there is a bit
    DelaySpraying : BOOL ;	//the analog value has change if there is a bit
    SpeedVentilatorBasicKiln : BOOL ;	//the analog value has change if there is a bit
    PositWasteAirFlapBasic : BOOL ;	//the analog value has change if there is a bit
    PositRecyclAirIFlapBasic : BOOL ;	//the analog value has change if there is a bit
    PositRecyclAirDFlapBasic : BOOL ;	//the analog value has change if there is a bit
    SpeedRotatingFloorDrives : BOOL ;	//the analog value has change if there is a bit
    spare_20 : BOOL ;
    spare_21 : BOOL ;
    spare_22 : BOOL ;
    spare_23 : BOOL ;
    spare_24 : BOOL ;
    spare_25 : BOOL ;
    spare_26 : BOOL ;
    spare_27 : BOOL ;
    spare_28 : BOOL ;
    spare_29 : BOOL ;
    spare_30 : BOOL ;
    spare_31 : BOOL ;
    spare_32 : BOOL ;
   END_STRUCT ;
  END_STRUCT ;	
END_TYPE

TYPE "SSA_Steep_Recipe_Header"	// UDT 2104
VERSION : 0.1
  STRUCT
   NumberOfSteps : INT  := 6;
   Steep_1_to_4 : DINT ;	//Byte 0 to 3 can be used to sign conical steeping vessel as used/not used
   Steep_5_to_6 : DINT ;	//Byte 0 to 3 can be used to sign conical steeping vessel as used/not used
   TemperaturAboveFloor : DINT ;	//Setpoint Temperature in °C (GMC)
   SPARE_DINT003 : DINT ;
   SPARE_DINT004 : DINT ;
   SPARE_DINT005 : DINT ;
   SPARE_DINT006 : DINT ;
   SPARE_INT000 : INT ;
   SPARE_INT001 : INT ;
   SPARE_INT002 : INT ;
   SPARE_INT003 : INT ;
   SPARE_INT004 : INT ;
   Loading : UDT 2011;
   Unloading : UDT 2012;
   Cleaning : UDT 2013;
  END_STRUCT ;	
END_TYPE

TYPE "SSA_Steep_Step"	// UDT 2105
VERSION : 0.1
  STRUCT
   StepNumber : INT  := 1;
   StepType : INT  := 1;	//Type Loading = 0;Wetsteep = 1;Drysteep = 2;unloading = 4;Cleaning = 8
   NextStep : INT  := 2;
   StepTime_Min : INT ;	//Minimal Steptime in min
   StepTime_Max : INT ;	//Maximal Steptime in min
   TemperaturWater : DINT ;	//Setpoint watertemperature in °C
   RecyclingWater : DINT ;	//Volume of water in m³
   FreshWater : DINT ;	//Volume of water in m³
   OffsetWater : DINT ;	//Volume of water in m³
   MinLevelWaterAeriation : DINT ;	//Volume of water in m³
   OverflowWater : DINT ;	//Volume of water in m³ (UAN)
   SprayDuringWaterFill : BYTE ;	//Spraying during fillup Water y/n (1/0)
   AeriationDuringWaterFill : BYTE ;	//Aeriation during fillup Water y/n (1/0)
   SprayDuringAeriation : BYTE ;	//Spraying during Aeriation y/n (1/0)to hold foam down
   CleaningSurface : BYTE ;	//Cleaning product surface y/n (1/0)
   AeriationConeNozzels : BYTE ;	//Aeriation during wetsteep via cone nozzles y/n (1/0) (UAN)
   AeriationHeinekenTube : BYTE ;	//Aeriation during wetsteep via Heinken Tube y/n (1/0) (UAN)
   WaterRecirculationContin : BYTE ;	//Continuesly water recirculation during wetsteep y/n (1/0) (UAN)
   WasteWaterToRecyclingTan : BYTE ;	//WasteWaterToRecyclingTank y/n (1/0) (YYR)
   Cooling : BYTE ;	//Activate Cooling System y/n (1/0) (GMC)
   AirMoisten : BYTE ;	//Moisten Air y/n (1/0) (GMC)
   NumberOfAeriationRounds : INT ;	//Number of Rounds of Aeriation
   NumberOfAeriationLines : INT ;	//Number of lines (valves) of Aeriation
   DelayNextValve : INT ;	//Delay to open next valve in sec (GMC)
   DelayNextAeriationCycle : INT ;	//Delay between two Aeriation-Starts in min/Aeriation time per tank (UAN)
   OverflowTime : INT ;	//Time to clean Surface in min(UAN)
   SpeedVentilator1 : INT ;	//Setpoint Fanspeed in % CO2 suck off Fan 1
   SpeedVentilator2 : INT ;	//Setpoint Fanspeed in % CO2 suck off Fan 2
   SpeedVentilator3 : INT ;	//Setpoint Fanspeed in % CO2 suck off Fan 3
   SpeedVentilator4 : INT ;	//Setpoint Fanspeed in % CO2 suck off Fan 4
   DrainTimeWaterAeriation : INT ;	//Time to drain Water before stop Aeriation in min
   DrainTimeWaterCO2Suck : INT ;	//Time to drain Water before Start CO2 suck off in min
   StartSpraying : INT ;	//Starttime spraying in min counted from start steptime
   TimeSpraying : INT ;	//Time one Round spraying
   DelaySpraying : INT ;	//Delay between two starts spraying
   PosExhaustAirFlapBasic : INT ;	//Setpoint basic flap position (GMC)
   DelayRecirculation : INT ;	//Delay to next run recirculation pump in min(UAN)
   TimeCO2Aeration : INT ;	//Time running CO2 Aeration
   DelayCO2Aeration : INT ;	//Delay between CO2 Aeration
   PumpP3_P4 : BYTE ;	//Pump 3 + P4 selected
   PumpP5_P6 : BYTE ;	//Pump 3 + P4 selected
   WaterRecirculationPeriod : BYTE ;	//Period. water recirculation during wetsteep y/n (1/0) (UAN)
   Spare : BYTE ;
   NoOfPulses : INT ;	//de: Anzahl_Takt
   SplitterBreak : INT ;	//de: Teiler_Pause
   TimeRecirculation : INT ;	//Time running recirculation pump in min(UAN)
  END_STRUCT ;	
END_TYPE

TYPE "SSA_Steep_Sum"	// UDT 2106
VERSION : 0.1
  STRUCT
   ActCondWaterVol_Saved : DINT ;	//Summary volume Conditioned water
   ActFreshWaterVol_Saved : DINT ;	//Summary volume Fresh water
   TimeCleanSurface : DINT ;	//Maximum Time to Clean Surface
   EdgeEvent2 : BOOL ;
   Profimess_Arbeit_Batch : REAL ;
   Value14 : DINT ;
  END_STRUCT ;	
END_TYPE

TYPE "SSA_Germ_Cmd"	// UDT 2200
VERSION : 0.1
  STRUCT
   Functions : STRUCT
    StartLoading : BOOL ;	//Start Function Loading
    BreakLoading : BOOL ;	//Break Function Loading
    ContinueLoading : BOOL ;	//Continue Function Loading
    StopLoading : BOOL ;	//Stop Function Loading
    UnloadingManuel : BOOL ;	//Unloading in Manuel Mode, only for Kiln
    StartUnloading : BOOL ;	//Start Function Unloading
    BreakUnloading : BOOL ;	//Break Function Unloading
    ContinueUnloading : BOOL ;	//Continue Function Unloading
    StopUnloading : BOOL ;	//Stop Function Unloading
    StartCleaning : BOOL ;	//Start Function Cleaning
    BreakCleaning : BOOL ;	//Break Function Cleaning
    ContinueCleaning : BOOL ;	//Continue Function Cleaning
    CleaningReady : BOOL ;	//Stop Function Cleaning
    StartProcess : BOOL ;	//Comand of Future
    Comand16 : BOOL ;
    Comand17 : BOOL ;
   END_STRUCT ;
   General : STRUCT
    LiftingDeviceUP : BOOL ;	//Lifting device UP
    LiftingDeviceDOWN : BOOL ;	//Lifting device DOWN
    LiftingDeviceSTOP : BOOL ;	//Lifting device STOP
    LiftingDeviceRESET : BOOL ;	//Lifting device RESET FAULT
    LoadUnloadScrewINSIDE : BOOL ;	//Loading-Unloading Screw INSIDE (LEFT)
    LoadUnloadScrewOUTSIDE : BOOL ;	//Loading-Unloading Screw OUTSIDE (RIGHT)
    LoadUnloadScrewSTOP : BOOL ;	//Loading-UnloadingScrew STOP
    LoadUnloadScrewRESET : BOOL ;	//Loading-UnloadingScrew RESET FAULT
    DischargeFlapOPEN : BOOL ;	//Discharge flap OPEN
    DischargeFlapCLOSE : BOOL ;	//Discharge flap CLOSE
    DischargeFlapRESET : BOOL ;	//Discharge flap RESET FAULT
    RotatingFloorDrivesRIGHT : BOOL ;	//Rotating Floor Drives RIGHT
    RotatingFloorDrivesLEFT : BOOL ;	//Rotating Floor Drives LEFT
    RotatingFloorDrivesSTOP : BOOL ;	//Rotating Floor Drives STOP
    RotatingFloorDrivesRESET : BOOL ;	//Rotating Floor Drives RESET FAULT
    spare_16 : BOOL ;
   END_STRUCT ;
   Germination : STRUCT
    TurningSpiralsSTART : BOOL ;	//Turning Spirals START
    TurningSpiralsSTOP : BOOL ;	//Turning Spirals STOP
    TurningSpiralsRESET : BOOL ;	//Turning Spirals RESET FAULT
    FloorCleanBelowSTART : BOOL ;	//START cleaning the floor from below
    FloorCleanBelowSTOP : BOOL ;	//STOP cleaning the floor from below
    FloorCleanBelowRESET : BOOL ;	//RESET FAULT cleaning the floor from below
    AirMoistenON : BOOL ;	//Air Moisten ON
    AirMoistenOFF : BOOL ;	//Air Moisten OFF
    AirMoistenRESET : BOOL ;	//Air Moisten RESET FAULT
    CoolingON : BOOL ;	//Cooling ON
    CoolingOFF : BOOL ;	//Cooling OFF
    CoolingRESET : BOOL ;	//Cooling RESET FAULT
    WallCleanBelowSTART : BOOL ;	//START cleaning wall below floor
    WallCleanBelowSTOP : BOOL ;	//STOP cleaning wall below floor
    WallCleanBelowRESET : BOOL ;	//RESET FAULT cleaning wall below floor
    WallCleanBelowSTART_L : BOOL ;	//START LEFT cleaning wall below floor
   END_STRUCT ;
   SPARE2 : BYTE ;
   SPARE3 : BYTE ;
   SPARE4 : BYTE ;
   SPARE5 : BYTE ;
  END_STRUCT ;	
END_TYPE

